ABB RAPID module: 000ACBDB

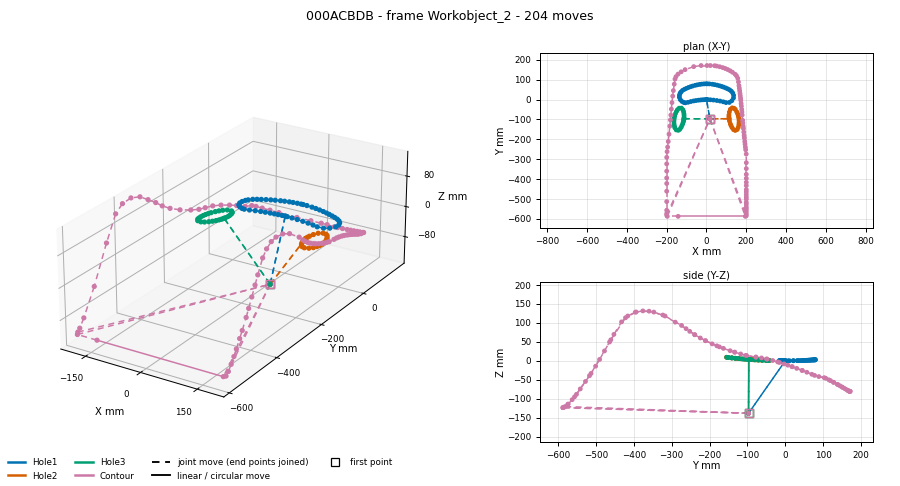
[picture p0: tool path of 000ACBDB in frame Workobject_2, 204 of 204 moves have a stored position in this frame; points joined in program order, loops and branches not executed]
MODULE Module1
        CONST robtarget Target_10:=[[26.851148837,-92.746056848,-137.743887933],[0.741188403,0.065864979,-0.059133334,0.6654358],[0,-1,-4,0],[9E+09,9E+09,9E+09,9E+09,9E+09,9E+09]];
    CONST robtarget H1_10:=[[5.822359777,-0.3029029,0.000239991],[0.999601623,-0.000118584,-0.000002778,-0.02822376],[0,-1,-1,0],[9E+09,9E+09,9E+09,9E+09,9E+09,9E+09]];
    CONST robtarget H1_20:=[[19.5237916,-1.229906178,0.000797071],[0.999216395,-0.000469719,-0.000020106,-0.039577455],[0,-1,0,0],[9E+09,9E+09,9E+09,9E+09,9E+09,9E+09]];
    CONST robtarget H1_30:=[[35.072112263,-2.692139723,0.003045649],[0.998507815,-0.001051706,-0.000057639,-0.054598844],[0,0,0,0],[9E+09,9E+09,9E+09,9E+09,9E+09,9E+09]];
    CONST robtarget H1_40:=[[51.872897494,-4.859700389,0.009441408],[0.997236669,-0.001878928,-0.000140271,-0.074266246],[0,0,0,0],[9E+09,9E+09,9E+09,9E+09,9E+09,9E+09]];
    CONST robtarget H1_50:=[[68.085842086,-7.671579778,0.023196339],[0.995164323,-0.002935794,-0.00030113,-0.098179733],[0,0,0,0],[9E+09,9E+09,9E+09,9E+09,9E+09,9E+09]];
    CONST robtarget H1_60:=[[84.016477696,-11.327527953,0.050315148],[0.991731899,-0.004378584,-0.000566998,-0.128251111],[0,0,0,0],[9E+09,9E+09,9E+09,9E+09,9E+09,9E+09]];
    CONST robtarget H1_70:=[[97.822312549,-15.342823644,0.092032674],[0.99493212,-0.005901634,-0.000604486,-0.100373712],[0,0,0,0],[9E+09,9E+09,9E+09,9E+09,9E+09,9E+09]];
    CONST robtarget H1_80:=[[114.627720719,-14.523229835,0.082502162],[0.982974748,-0.00555832,0.001038246,0.183653673],[0,0,0,0],[9E+09,9E+09,9E+09,9E+09,9E+09,9E+09]];
    CONST robtarget H1_90:=[[127.080680914,-6.164946714,0.015071505],[0.921910532,-0.002219077,0.0009341,0.387395372],[0,0,0,0],[9E+09,9E+09,9E+09,9E+09,9E+09,9E+09]];
    CONST robtarget H1_100:=[[135.46672126,7.649000487,0.023178554],[0.80179062,0.002410603,-0.00179684,0.597597492],[0,0,0,0],[9E+09,9E+09,9E+09,9E+09,9E+09,9E+09]];
    CONST robtarget H1_110:=[[136.157764084,21.042101165,0.174701099],[0.644801471,0.005362679,-0.006356556,0.764304847],[0,0,0,0],[9E+09,9E+09,9E+09,9E+09,9E+09,9E+09]];
    CONST robtarget H1_120:=[[131.874650789,32.837383759,0.404255936],[0.501756468,0.004666505,-0.008044466,0.864958934],[0,0,0,0],[9E+09,9E+09,9E+09,9E+09,9E+09,9E+09]];
    CONST robtarget H1_130:=[[124.935320592,41.709089606,0.620811537],[0.38373825,0.005805796,-0.013969102,0.923317991],[0,0,0,0],[9E+09,9E+09,9E+09,9E+09,9E+09,9E+09]];
    CONST robtarget H1_140:=[[116.229745208,48.490778985,0.856866002],[0.260536152,0.005127658,-0.018998209,0.965263533],[0,0,0,0],[9E+09,9E+09,9E+09,9E+09,9E+09,9E+09]];
    CONST robtarget H1_150:=[[106.531812126,53.651183132,1.078234714],[0.225840714,0.005240396,-0.022598239,0.973887997],[0,0,0,0],[9E+09,9E+09,9E+09,9E+09,9E+09,9E+09]];
    CONST robtarget H1_160:=[[96.895202054,58.051394326,1.295938149],[0.200438859,0.005260811,-0.025705853,0.979354786],[0,0,0,0],[9E+09,9E+09,9E+09,9E+09,9E+09,9E+09]];
    CONST robtarget H1_170:=[[86.200217498,62.31165247,1.532433666],[0.177271875,0.005181025,-0.02875481,0.983728113],[0,0,0,0],[9E+09,9E+09,9E+09,9E+09,9E+09,9E+09]];
    CONST robtarget H1_180:=[[76.71572938,65.636541326,1.734823668],[0.158973824,0.005020732,-0.031165772,0.986777994],[0,0,0,0],[9E+09,9E+09,9E+09,9E+09,9E+09,9E+09]];
    CONST robtarget H1_190:=[[65.746053731,69.013152347,1.956481108],[0.13904105,0.004727267,-0.033645532,0.989703601],[0,0,0,0],[9E+09,9E+09,9E+09,9E+09,9E+09,9E+09]];
    CONST robtarget H1_200:=[[53.528960273,72.219165213,2.182137232],[0.117236878,0.004256713,-0.036032694,0.99244095],[0,0,0,0],[9E+09,9E+09,9E+09,9E+09,9E+09,9E+09]];
    CONST robtarget H1_210:=[[41.391728548,74.836405126,2.377436106],[0.09495427,0.003628233,-0.038009225,0.994749125],[0,0,0,0],[9E+09,9E+09,9E+09,9E+09,9E+09,9E+09]];
    CONST robtarget H1_220:=[[29.543599616,76.831762317,2.533066199],[0.071726163,0.002844733,-0.039536532,0.996636407],[0,0,0,0],[9E+09,9E+09,9E+09,9E+09,9E+09,9E+09]];
    CONST robtarget H1_230:=[[14.423984972,78.513378499,2.668784241],[0.038405498,0.001570062,-0.040842603,0.998425978],[0,0,0,0],[9E+09,9E+09,9E+09,9E+09,9E+09,9E+09]];
    CONST robtarget H1_240:=[[3.529088415,79.053026073,2.713218089],[0.010521449,0.000436179,-0.041267795,0.999092627],[0,0,0,0],[9E+09,9E+09,9E+09,9E+09,9E+09,9E+09]];
    CONST robtarget H1_250:=[[-2.41393131,79.072935695,2.714873077],[0.007473374,0.000309011,0.041283579,-0.999119472],[-1,0,-2,0],[9E+09,9E+09,9E+09,9E+09,9E+09,9E+09]];
    CONST robtarget H1_260:=[[-12.79429846,78.631983773,2.678514834],[0.034459184,0.001412549,0.040935724,-0.99856639],[-1,0,-2,0],[9E+09,9E+09,9E+09,9E+09,9E+09,9E+09]];
    CONST robtarget H1_270:=[[-24.249294402,77.535857479,2.589375882],[0.060604597,0.002435338,0.04008087,-0.997353837],[-1,0,-2,0],[9E+09,9E+09,9E+09,9E+09,9E+09,9E+09]];
    CONST robtarget H1_280:=[[-34.022487008,76.144299483,2.478783806],[0.080709455,0.003161608,0.039008163,-0.995969051],[-1,0,-2,0],[9E+09,9E+09,9E+09,9E+09,9E+09,9E+09]];
    CONST robtarget H1_290:=[[-46.078360434,73.893089687,2.305893098],[0.103704766,0.003891012,0.037293549,-0.993901088],[-1,0,-2,0],[9E+09,9E+09,9E+09,9E+09,9E+09,9E+09]];
    CONST robtarget H1_300:=[[-56.338244037,71.532430973,2.132551125],[0.12227693,0.004378833,0.035518358,-0.991850606],[-1,0,-2,0],[9E+09,9E+09,9E+09,9E+09,9E+09,9E+09]];
    CONST robtarget H1_310:=[[-69.339991697,67.960014478,1.885584593],[0.145492672,0.004836435,0.032868463,-0.988801373],[-1,0,-2,0],[9E+09,9E+09,9E+09,9E+09,9E+09,9E+09]];
    CONST robtarget H1_320:=[[-80.066156183,64.506655976,1.664288351],[0.165267796,0.005087248,0.030343309,-0.985768715],[-1,0,-2,0],[9E+09,9E+09,9E+09,9E+09,9E+09,9E+09]];
    CONST robtarget H1_330:=[[-91.064867974,60.445719882,1.42572312],[0.187354774,0.005230691,0.027414242,-0.981895762],[-1,0,-2,0],[9E+09,9E+09,9E+09,9E+09,9E+09,9E+09]];
    CONST robtarget H1_340:=[[-101.905940758,55.839614159,1.18312319],[0.212963875,0.005260152,0.02413793,-0.976747705],[-1,0,-2,0],[9E+09,9E+09,9E+09,9E+09,9E+09,9E+09]];
    CONST robtarget H1_350:=[[-111.354611608,51.195431258,0.968343063],[0.241468672,0.005196012,0.020879464,-0.970170052],[-1,0,-2,0],[9E+09,9E+09,9E+09,9E+09,9E+09,9E+09]];
    CONST robtarget H1_360:=[[-120.397291393,45.950711286,0.761205788],[0.279512614,0.005021911,0.017247524,-0.959973959],[-1,0,-2,0],[9E+09,9E+09,9E+09,9E+09,9E+09,9E+09]];
    CONST robtarget H1_370:=[[-128.598391018,37.638733053,0.508601596],[0.433495604,0.005392781,0.011207446,-0.901069849],[-1,0,-2,0],[9E+09,9E+09,9E+09,9E+09,9E+09,9E+09]];
    CONST robtarget H1_380:=[[-132.59535291,31.513908724,0.380771009],[0.519470782,0.004385873,0.007214063,-0.854446504],[-1,0,-2,0],[9E+09,9E+09,9E+09,9E+09,9E+09,9E+09]];
    CONST robtarget H1_390:=[[-136.029541122,21.745014519,0.186590065],[0.636693593,0.005473624,0.006628875,-0.771068977],[-1,0,-2,0],[9E+09,9E+09,9E+09,9E+09,9E+09,9E+09]];
    CONST robtarget H1_400:=[[-136.249962901,11.059124977,0.04827139],[0.761868919,0.003316184,0.002819313,-0.647716609],[-1,0,-2,0],[9E+09,9E+09,9E+09,9E+09,9E+09,9E+09]];
    CONST robtarget H1_410:=[[-131.64005613,-0.499314804,0.000306325],[0.879140299,-0.000171436,-0.000093084,-0.476563004],[-1,0,-2,0],[9E+09,9E+09,9E+09,9E+09,9E+09,9E+09]];
    CONST robtarget H1_420:=[[-123.455867891,-9.420071732,0.0348798],[0.944806429,-0.003471167,-0.00120507,-0.327608472],[0,0,0,0],[9E+09,9E+09,9E+09,9E+09,9E+09,9E+09]];
    CONST robtarget H1_430:=[[-113.576963132,-14.907418805,0.086903996],[0.986261821,-0.005723499,-0.000957591,-0.165087688],[0,0,0,0],[9E+09,9E+09,9E+09,9E+09,9E+09,9E+09]];
    CONST robtarget H1_440:=[[-106.317369492,-16.310941036,0.103957245],[0.999811227,-0.006344693,-0.000116729,-0.018364159],[0,0,0,0],[9E+09,9E+09,9E+09,9E+09,9E+09,9E+09]];
    CONST robtarget H1_450:=[[-92.832473373,-13.839947638,0.074955681],[0.988817126,-0.005329902,0.000803336,0.149035693],[0,0,0,0],[9E+09,9E+09,9E+09,9E+09,9E+09,9E+09]];
    CONST robtarget H1_460:=[[-78.807083419,-10.018549669,0.039414696],[0.993068241,-0.003881094,0.000459005,0.117474235],[0,0,0,0],[9E+09,9E+09,9E+09,9E+09,9E+09,9E+09]];
    CONST robtarget H1_470:=[[-65.187150671,-7.109105356,0.019965876],[0.995622128,-0.00276447,0.000259127,0.093428411],[0,0,0,0],[9E+09,9E+09,9E+09,9E+09,9E+09,9E+09]];
    CONST robtarget H1_480:=[[-53.308517932,-5.077796928,0.010293707],[0.99709043,-0.001979187,0.000151084,0.076201937],[0,0,0,0],[9E+09,9E+09,9E+09,9E+09,9E+09,9E+09]];
    CONST robtarget H2_10:=[[113.353839197,-96.530340155,3.554586283],[0.748476702,-0.027164205,-0.024031886,-0.66216856],[0,-2,0,0],[9E+09,9E+09,9E+09,9E+09,9E+09,9E+09]];
    CONST robtarget H2_20:=[[115.464244857,-108.261236654,4.456832066],[0.783370795,-0.031725245,-0.025118376,-0.620236063],[0,-2,0,0],[9E+09,9E+09,9E+09,9E+09,9E+09,9E+09]];
    CONST robtarget H2_30:=[[119.841770859,-122.609627571,5.694437701],[0.820338947,-0.037394525,-0.025986049,-0.570061739],[0,-2,0,0],[9E+09,9E+09,9E+09,9E+09,9E+09,9E+09]];
    CONST robtarget H2_40:=[[123.527187524,-131.471644624,6.531828825],[0.840093436,-0.040906802,-0.026306691,-0.540256985],[0,-2,0,0],[9E+09,9E+09,9E+09,9E+09,9E+09,9E+09]];
    CONST robtarget H2_50:=[[128.497488384,-141.378498828,7.628466543],[0.858996843,-0.051948016,-0.030746201,-0.508409774],[0,-2,0,0],[9E+09,9E+09,9E+09,9E+09,9E+09,9E+09]];
    CONST robtarget H2_60:=[[136.105023801,-151.417458815,8.807259628],[0.9370628,-0.052968209,-0.019477183,-0.344569757],[0,-2,1,0],[9E+09,9E+09,9E+09,9E+09,9E+09,9E+09]];
    CONST robtarget H2_70:=[[144.44174435,-155.241358627,9.235032257],[0.998005294,-0.054882138,-0.001713201,-0.031152033],[0,-2,1,0],[9E+09,9E+09,9E+09,9E+09,9E+09,9E+09]];
    CONST robtarget H2_80:=[[154.006118475,-150.661083946,8.721245568],[0.908752155,-0.051640643,0.023496208,0.41346184],[0,-2,-2,0],[9E+09,9E+09,9E+09,9E+09,9E+09,9E+09]];
    CONST robtarget H2_90:=[[159.658512318,-139.997126678,7.46002746],[0.79556302,-0.048534782,0.036779081,0.60280275],[0,-2,-2,0],[9E+09,9E+09,9E+09,9E+09,9E+09,9E+09]];
    CONST robtarget H2_100:=[[162.376179916,-127.516765295,6.151270714],[0.758777117,-0.035896886,0.030733454,0.649633862],[0,-2,-2,0],[9E+09,9E+09,9E+09,9E+09,9E+09,9E+09]];
    CONST robtarget H2_110:=[[163.475309343,-117.188024925,5.209561495],[0.726089453,-0.031708487,0.029967159,0.686214724],[0,-2,-2,0],[9E+09,9E+09,9E+09,9E+09,9E+09,9E+09]];
    CONST robtarget H2_120:=[[163.492051849,-105.498676679,4.235442415],[0.68742213,-0.02716136,0.028653424,0.725184154],[0,-2,-2,0],[9E+09,9E+09,9E+09,9E+09,9E+09,9E+09]];
    CONST robtarget H2_130:=[[162.227653576,-93.852494517,3.362554996],[0.647198475,-0.022863035,0.026901004,0.761503612],[0,-2,-2,0],[9E+09,9E+09,9E+09,9E+09,9E+09,9E+09]];
    CONST robtarget H2_140:=[[160.115266627,-83.883832167,2.693495802],[0.611329591,-0.019384569,0.025073576,0.790741226],[0,-2,-2,0],[9E+09,9E+09,9E+09,9E+09,9E+09,9E+09]];
    CONST robtarget H2_150:=[[156.297628088,-71.997621841,1.990746535],[0.566564132,-0.015498139,0.022528309,0.823563821],[0,-2,-2,0],[9E+09,9E+09,9E+09,9E+09,9E+09,9E+09]];
    CONST robtarget H2_160:=[[151.695554905,-61.57696201,1.460402668],[0.525052814,-0.012338693,0.019992429,0.850745321],[0,-2,-2,0],[9E+09,9E+09,9E+09,9E+09,9E+09,9E+09]];
    CONST robtarget H2_170:=[[144.697582417,-49.505236902,0.947141756],[0.473504531,-0.008991922,0.016722668,0.880586711],[0,-2,-2,0],[9E+09,9E+09,9E+09,9E+09,9E+09,9E+09]];
    CONST robtarget H2_180:=[[138.479508342,-43.903121696,0.746107759],[0.27767732,-0.00468769,0.016215326,0.960526103],[0,-2,-2,0],[9E+09,9E+09,9E+09,9E+09,9E+09,9E+09]];
    CONST robtarget H2_190:=[[129.228972872,-41.777368956,0.676021991],[0.096272542,-0.00154838,-0.016002122,-0.995225167],[0,-2,-1,0],[9E+09,9E+09,9E+09,9E+09,9E+09,9E+09]];
    CONST robtarget H2_200:=[[119.969352837,-48.884343518,0.92369665],[0.471525813,-0.008844606,-0.016537415,-0.88165282],[0,-2,-1,0],[9E+09,9E+09,9E+09,9E+09,9E+09,9E+09]];
    CONST robtarget H2_210:=[[114.862919521,-62.738334039,1.515519436],[0.627584743,-0.01501889,-0.018622826,-0.778180579],[0,-2,0,0],[9E+09,9E+09,9E+09,9E+09,9E+09,9E+09]];
    CONST robtarget H2_220:=[[112.782345249,-77.613018099,2.309812122],[0.68393145,-0.020117567,-0.021445948,-0.728953446],[0,-2,0,0],[9E+09,9E+09,9E+09,9E+09,9E+09,9E+09]];
    CONST robtarget H2_230:=[[112.619785188,-86.868177001,2.886201345],[0.71669986,-0.023502264,-0.022847584,-0.69661104],[0,-2,0,0],[9E+09,9E+09,9E+09,9E+09,9E+09,9E+09]];
    CONST robtarget H2_240:=[[-146.211495519,-51.850497933,1.03831773],[0.483686197,-0.009610968,-0.017386784,-0.875015995],[0,0,0,0],[9E+09,9E+09,9E+09,9E+09,9E+09,9E+09]];
    CONST robtarget H2_250:=[[-149.107034596,-56.713931894,1.240531943],[0.504739909,-0.010947301,-0.018717571,-0.862999092],[0,0,0,0],[9E+09,9E+09,9E+09,9E+09,9E+09,9E+09]];
    CONST robtarget H2_260:=[[-151.196381116,-60.595266341,1.414599226],[0.521004601,-0.012053404,-0.019739665,-0.853240451],[0,0,0,0],[9E+09,9E+09,9E+09,9E+09,9E+09,9E+09]];
    CONST robtarget H2_270:=[[-153.664684888,-65.700778492,1.660655818],[0.541786795,-0.013561095,-0.021028685,-0.840143416],[0,0,0,0],[9E+09,9E+09,9E+09,9E+09,9E+09,9E+09]];
    CONST robtarget H2_280:=[[-155.154121582,-69.132687567,1.836925418],[0.555398018,-0.014605886,-0.021858445,-0.831169007],[0,0,0,0],[9E+09,9E+09,9E+09,9E+09,9E+09,9E+09]];
    CONST robtarget H2_290:=[[-156.838393073,-73.438168646,2.070385804],[0.572126761,-0.015952496,-0.022858608,-0.819691388],[0,0,0,0],[9E+09,9E+09,9E+09,9E+09,9E+09,9E+09]];
    CONST robtarget H2_300:=[[-158.385938506,-77.933906529,2.328748906],[0.589243008,-0.01740327,-0.023847263,-0.807416318],[0,0,0,0],[9E+09,9E+09,9E+09,9E+09,9E+09,9E+09]];
    CONST robtarget H2_310:=[[-159.957660119,-83.287580126,2.655778618],[0.609137583,-0.019181563,-0.024956614,-0.792439676],[0,0,0,0],[9E+09,9E+09,9E+09,9E+09,9E+09,9E+09]];
    CONST robtarget H2_320:=[[-160.980080082,-87.442702976,2.924049197],[0.624309267,-0.020604348,-0.025759704,-0.780480517],[0,0,0,0],[9E+09,9E+09,9E+09,9E+09,9E+09,9E+09]];
    CONST robtarget H2_330:=[[-161.982296625,-92.416885735,3.261751009],[0.642117861,-0.022350365,-0.026655965,-0.765816279],[0,0,0,0],[9E+09,9E+09,9E+09,9E+09,9E+09,9E+09]];
    CONST robtarget H2_340:=[[-162.658869303,-96.728725981,3.569023092],[0.657295549,-0.023901838,-0.027373156,-0.752756252],[0,0,0,0],[9E+09,9E+09,9E+09,9E+09,9E+09,9E+09]];
    CONST robtarget H2_350:=[[-163.3089721,-102.754467741,4.020957585],[0.678104452,-0.026127054,-0.028278994,-0.73395642],[0,0,0,0],[9E+09,9E+09,9E+09,9E+09,9E+09,9E+09]];
    CONST robtarget H2_360:=[[-163.588731895,-107.752945715,4.415691555],[0.695018407,-0.028020761,-0.028942698,-0.717862501],[0,0,0,0],[9E+09,9E+09,9E+09,9E+09,9E+09,9E+09]];
    CONST robtarget H2_370:=[[-163.618228194,-113.559417795,4.896727938],[0.714282559,-0.030273854,-0.029608796,-0.698575149],[0,0,0,0],[9E+09,9E+09,9E+09,9E+09,9E+09,9E+09]];
    CONST robtarget H2_380:=[[-163.400274185,-118.383550137,5.314692806],[0.729948009,-0.032185694,-0.030075106,-0.68208172],[0,0,0,0],[9E+09,9E+09,9E+09,9E+09,9E+09,9E+09]];
    CONST robtarget H2_390:=[[-162.725296292,-125.102597289,5.924399836],[0.751271747,-0.034905156,-0.030588292,-0.658359133],[0,0,0,0],[9E+09,9E+09,9E+09,9E+09,9E+09,9E+09]];
    CONST robtarget H2_400:=[[-161.284238305,-133.391691812,6.720562185],[0.776702072,-0.038351334,-0.030988752,-0.627935318],[0,0,0,0],[9E+09,9E+09,9E+09,9E+09,9E+09,9E+09]];
    CONST robtarget H2_410:=[[-159.646201857,-140.03915335,7.465181503],[0.795699451,-0.048528933,-0.036759329,-0.602624326],[0,0,0,0],[9E+09,9E+09,9E+09,9E+09,9E+09,9E+09]];
    CONST robtarget H2_420:=[[-157.038646765,-146.326115351,8.219442761],[0.863010837,-0.050522948,-0.029376394,-0.501793537],[0,0,0,0],[9E+09,9E+09,9E+09,9E+09,9E+09,9E+09]];
    CONST robtarget H2_430:=[[-154.143947087,-150.501789747,8.703078987],[0.906591242,-0.051576054,-0.023790201,-0.418170129],[0,0,0,0],[9E+09,9E+09,9E+09,9E+09,9E+09,9E+09]];
    CONST robtarget H2_440:=[[-151.052306188,-153.326067118,9.022258344],[0.953526504,-0.053170779,-0.016512614,-0.296120598],[0,0,0,0],[9E+09,9E+09,9E+09,9E+09,9E+09,9E+09]];
    CONST robtarget H2_450:=[[-147.24920751,-155.018200209,9.210400641],[0.992262537,-0.054655516,-0.006130652,-0.111311491],[-1,1,-2,0],[9E+09,9E+09,9E+09,9E+09,9E+09,9E+09]];
    CONST robtarget H2_460:=[[-141.774746784,-154.730898904,9.178619755],[0.986433645,-0.054448707,0.008535421,0.154632303],[-1,1,-2,0],[9E+09,9E+09,9E+09,9E+09,9E+09,9E+09]];
    CONST robtarget H2_470:=[[-137.124498645,-152.232288983,8.899410279],[0.946429998,-0.053189584,0.017871487,0.317996442],[-1,1,-2,0],[9E+09,9E+09,9E+09,9E+09,9E+09,9E+09]];
    CONST robtarget H2_480:=[[-133.464165375,-148.877446335,8.516599917],[0.914460182,-0.052613853,0.02304735,0.400578554],[-1,1,-2,0],[9E+09,9E+09,9E+09,9E+09,9E+09,9E+09]];
    CONST robtarget H2_490:=[[-130.178716496,-144.342311293,7.984808374],[0.86461459,-0.051289546,0.029597151,0.498933866],[0,0,0,0],[9E+09,9E+09,9E+09,9E+09,9E+09,9E+09]];
    CONST robtarget H2_500:=[[-127.259861509,-139.094676901,7.34918768],[0.854541306,-0.052433266,0.031646215,0.515760047],[0,0,0,0],[9E+09,9E+09,9E+09,9E+09,9E+09,9E+09]];
    CONST robtarget H2_510:=[[-126.560241996,-137.75989446,7.184074667],[0.851876838,-0.052707296,0.032178927,0.520088753],[0,0,0,0],[9E+09,9E+09,9E+09,9E+09,9E+09,9E+09]];
    CONST robtarget H2_520:=[[-124.896955353,-134.374624635,6.818180126],[0.846081591,-0.042055694,0.026381033,0.530736565],[0,0,0,0],[9E+09,9E+09,9E+09,9E+09,9E+09,9E+09]];
    CONST robtarget H2_530:=[[-122.756510357,-129.759645709,6.365744431],[0.836453631,-0.040228874,0.026256095,0.545928181],[0,0,0,0],[9E+09,9E+09,9E+09,9E+09,9E+09,9E+09]];
    CONST robtarget H3_90:=[[-151.032520543,-60.277726678,1.399936408],[0.519689718,-0.011961435,-0.019657661,-0.854045138],[-1,1,1,0],[9E+09,9E+09,9E+09,9E+09,9E+09,9E+09]];
    CONST robtarget H3_100:=[[-155.411707479,-69.759012426,1.870035967],[0.557852374,-0.014799042,-0.022007461,-0.829516358],[-1,1,1,0],[9E+09,9E+09,9E+09,9E+09,9E+09,9E+09]];
    CONST robtarget H3_110:=[[-159.625213408,-82.068644739,2.579473667],[0.604642285,-0.018772206,-0.024709982,-0.79589241],[-1,1,1,0],[9E+09,9E+09,9E+09,9E+09,9E+09,9E+09]];
    CONST robtarget H3_120:=[[-161.878029858,-91.838551641,3.22156317],[0.640063811,-0.022144937,-0.026555455,-0.767543306],[-1,1,1,0],[9E+09,9E+09,9E+09,9E+09,9E+09,9E+09]];
    CONST robtarget H3_130:=[[-163.203180759,-101.514565736,3.925825431],[0.673850412,-0.025662667,-0.028101558,-0.737887087],[-1,1,1,0],[9E+09,9E+09,9E+09,9E+09,9E+09,9E+09]];
    CONST robtarget H3_140:=[[-163.644574839,-111.272609544,4.704398344],[0.706753039,-0.029380699,-0.02935936,-0.706240005],[-1,1,1,0],[9E+09,9E+09,9E+09,9E+09,9E+09,9E+09]];
    CONST robtarget H3_150:=[[-163.073115646,-122.1735858,5.654675757],[0.742058033,-0.033712272,-0.030383983,-0.668797556],[-1,1,1,0],[9E+09,9E+09,9E+09,9E+09,9E+09,9E+09]];
    CONST robtarget H3_160:=[[-161.45041585,-132.605221729,6.642943788],[0.774331563,-0.038018965,-0.030963091,-0.630877544],[0,0,0,0],[9E+09,9E+09,9E+09,9E+09,9E+09,9E+09]];
    CONST robtarget H3_170:=[[-159.100531555,-141.897037426,7.691315566],[0.801095296,-0.048179165,-0.035972301,-0.5955091],[0,0,0,0],[9E+09,9E+09,9E+09,9E+09,9E+09,9E+09]];
    CONST robtarget H3_180:=[[-152.159173857,-152.48346178,8.927706865],[0.937417285,-0.05258876,-0.01927966,-0.34367361],[0,0,0,0],[9E+09,9E+09,9E+09,9E+09,9E+09,9E+09]];
    CONST robtarget H3_190:=[[-141.819169103,-154.744996081,9.180180698],[0.986731419,-0.054459539,0.008429136,0.152722671],[-1,1,-2,0],[9E+09,9E+09,9E+09,9E+09,9E+09,9E+09]];
    CONST robtarget H3_200:=[[-134.593857995,-150.038962909,8.65016057],[0.923763552,-0.052723447,0.021614172,0.378700364],[-1,1,-2,0],[9E+09,9E+09,9E+09,9E+09,9E+09,9E+09]];
    CONST robtarget H3_210:=[[-128.24945161,-140.928737155,7.573794657],[0.858129871,-0.052045202,0.030922266,0.509851189],[0,0,0,0],[9E+09,9E+09,9E+09,9E+09,9E+09,9E+09]];
    CONST robtarget H3_220:=[[-123.697125678,-131.841961932,6.568031258],[0.840871704,-0.041053612,0.026317047,0.539033201],[0,0,0,0],[9E+09,9E+09,9E+09,9E+09,9E+09,9E+09]];
    CONST robtarget H3_230:=[[-119.718209049,-122.278505657,5.664229892],[0.819556015,-0.037263357,0.025971018,0.571196014],[0,0,0,0],[9E+09,9E+09,9E+09,9E+09,9E+09,9E+09]];
    CONST robtarget H3_240:=[[-116.914843491,-113.780868438,4.915548572],[0.79834197,-0.033899897,0.025507908,0.600708118],[0,0,0,0],[9E+09,9E+09,9E+09,9E+09,9E+09,9E+09]];
    CONST robtarget H3_250:=[[-115.129078785,-106.801898067,4.339203478],[0.779261299,-0.031153062,0.025003039,0.625424786],[0,0,0,0],[9E+09,9E+09,9E+09,9E+09,9E+09,9E+09]];
    CONST robtarget H3_260:=[[-113.89814797,-100.37190359,3.839131682],[0.760357658,-0.02864585,0.024428314,0.648412603],[0,0,0,0],[9E+09,9E+09,9E+09,9E+09,9E+09,9E+09]];
    CONST robtarget H3_270:=[[-2.8649147,79.065647891,2.714269653],[0.008725056,0.000360634,0.041277791,-0.999109547],[0,0,0,0],[9E+09,9E+09,9E+09,9E+09,9E+09,9E+09]];
    CONST robtarget H3_280:=[[-6.334685984,78.972502416,2.706566926],[0.018106651,0.000746596,0.041203984,-0.998986398],[-1,0,-2,0],[9E+09,9E+09,9E+09,9E+09,9E+09,9E+09]];
    CONST robtarget H3_290:=[[-10.115541125,78.798786754,2.692234704],[0.027838843,0.001144817,0.041066905,-0.99876784],[-1,0,-2,0],[9E+09,9E+09,9E+09,9E+09,9E+09,9E+09]];
    CONST robtarget H3_300:=[[-12.967121471,78.620009059,2.677531525],[0.034878932,0.001429434,0.040926321,-0.998552178],[-1,0,-2,0],[9E+09,9E+09,9E+09,9E+09,9E+09,9E+09]];
    CONST robtarget H3_310:=[[-17.148960654,78.286603961,2.650238016],[0.044763067,0.001824202,0.040665248,-0.998167961],[-1,0,-2,0],[9E+09,9E+09,9E+09,9E+09,9E+09,9E+09]];
    CONST robtarget H3_320:=[[-21.565389337,77.846298964,2.614439805],[0.054738413,0.002212749,0.040322016,-0.99768379],[-1,0,-2,0],[9E+09,9E+09,9E+09,9E+09,9E+09,9E+09]];
    CONST robtarget H3_330:=[[-27.10271187,77.171238947,2.56012345],[0.066674643,0.002660905,0.039798533,-0.996977175],[-1,0,-2,0],[9E+09,9E+09,9E+09,9E+09,9E+09,9E+09]];
    CONST robtarget H3_340:=[[-30.430871342,76.702094493,2.522774606],[0.073533349,0.002909696,0.039436657,-0.99650847],[-1,0,-2,0],[9E+09,9E+09,9E+09,9E+09,9E+09,9E+09]];
    CONST robtarget H3_350:=[[-36.071948771,75.802452022,2.452048787],[0.084738305,0.003298132,0.038746269,-0.995644148],[-1,0,-2,0],[9E+09,9E+09,9E+09,9E+09,9E+09,9E+09]];
    CONST robtarget H3_360:=[[-40.871398594,74.935924168,2.385053721],[0.093983304,0.003597617,0.038084851,-0.99483855],[-1,0,-2,0],[9E+09,9E+09,9E+09,9E+09,9E+09,9E+09]];
    CONST robtarget H3_370:=[[-45.168917683,74.082828858,2.320177807],[0.102030362,0.003842105,0.03743714,-0.994069165],[-1,0,-2,0],[9E+09,9E+09,9E+09,9E+09,9E+09,9E+09]];
    CONST robtarget H3_380:=[[-50.551705589,72.913466151,2.232974457],[0.111870475,0.004118016,0.036554348,-0.9930417],[-1,0,-2,0],[9E+09,9E+09,9E+09,9E+09,9E+09,9E+09]];
    CONST robtarget H3_390:=[[-55.549209342,71.72828369,2.146624137],[0.12086579,0.004345406,0.035664857,-0.992018445],[-1,0,-2,0],[9E+09,9E+09,9E+09,9E+09,9E+09,9E+09]];
    CONST robtarget H3_400:=[[-61.927505303,70.076739745,2.029695738],[0.132245008,0.004596819,0.034433562,-0.990608125],[-1,0,-2,0],[9E+09,9E+09,9E+09,9E+09,9E+09,9E+09]];
    CONST robtarget H3_410:=[[-68.62429444,68.173796841,1.899846076],[0.144200224,0.004815742,0.033025964,-0.988985536],[-1,0,-2,0],[9E+09,9E+09,9E+09,9E+09,9E+09,9E+09]];
    CONST robtarget H3_420:=[[-73.053957234,66.817667973,1.810494492],[0.152245741,0.004935728,0.032029173,-0.987811219],[-1,0,-2,0],[9E+09,9E+09,9E+09,9E+09,9E+09,9E+09]];
    CONST robtarget H3_430:=[[-79.167968195,64.814210939,1.683307668],[0.163563945,0.005070503,0.030566866,-0.98604604],[-1,0,-2,0],[9E+09,9E+09,9E+09,9E+09,9E+09,9E+09]];
    CONST robtarget H3_440:=[[-84.238390617,63.031729667,1.574946041],[0.173348853,0.005155043,0.029274559,-0.984411804],[-1,0,-2,0],[9E+09,9E+09,9E+09,9E+09,9E+09,9E+09]];
    CONST robtarget H3_450:=[[-88.890544547,61.293706375,1.47361581],[0.182762993,0.005211361,0.028022536,-0.982743745],[-1,0,-2,0],[9E+09,9E+09,9E+09,9E+09,9E+09,9E+09]];
    CONST robtarget H3_460:=[[-95.479750625,58.649863335,1.327607794],[0.197052537,0.005258002,0.026132891,-0.980030471],[-1,0,-2,0],[9E+09,9E+09,9E+09,9E+09,9E+09,9E+09]];
    CONST robtarget H3_470:=[[-102.280879458,55.667700917,1.174643979],[0.213962984,0.0052591,0.024016447,-0.976532331],[-1,0,-2,0],[9E+09,9E+09,9E+09,9E+09,9E+09,9E+09]];
    CONST robtarget H3_480:=[[-108.13915594,52.85405221,1.041654244],[0.230734556,0.005228689,0.022039645,-0.972753042],[-1,0,-2,0],[9E+09,9E+09,9E+09,9E+09,9E+09,9E+09]];
    CONST robtarget H3_490:=[[-112.844891048,50.394720403,0.934303108],[0.246880393,0.005177668,0.020321316,-0.968819027],[-1,0,-2,0],[9E+09,9E+09,9E+09,9E+09,9E+09,9E+09]];
    CONST robtarget H3_500:=[[-118.347328888,47.230096261,0.808297005],[0.270328919,0.005090046,0.018124474,-0.962583955],[-1,0,-2,0],[9E+09,9E+09,9E+09,9E+09,9E+09,9E+09]];
    CONST robtarget H3_510:=[[-123.252061757,43.344922201,0.672097613],[0.369331386,0.005987744,0.015069422,-0.929156277],[-1,0,-2,0],[9E+09,9E+09,9E+09,9E+09,9E+09,9E+09]];
    CONST robtarget H3_520:=[[-127.934077654,38.449353154,0.529203927],[0.422392751,0.005479549,0.011756156,-0.906320104],[-1,0,-2,0],[9E+09,9E+09,9E+09,9E+09,9E+09,9E+09]];
    CONST robtarget H3_530:=[[-130.333027831,35.297380543,0.453953091],[0.466730019,0.005087182,0.009640709,-0.884332667],[-1,0,-2,0],[9E+09,9E+09,9E+09,9E+09,9E+09,9E+09]];
    CONST robtarget H3_540:=[[-132.17837315,32.294925109,0.39435499],[0.509131796,0.004556015,0.007701531,-0.860642053],[-1,0,-2,0],[9E+09,9E+09,9E+09,9E+09,9E+09,9E+09]];
    CONST robtarget H3_550:=[[-134.71177698,26.636386283,0.280260541],[0.579626455,0.006116566,0.008598406,-0.814813984],[-1,0,-2,0],[9E+09,9E+09,9E+09,9E+09,9E+09,9E+09]];
    CONST robtarget H3_560:=[[-135.896350855,22.401538281,0.198051061],[0.629116362,0.005573246,0.006885644,-0.777260657],[-1,0,-2,0],[9E+09,9E+09,9E+09,9E+09,9E+09,9E+09]];
    CONST robtarget H3_570:=[[-136.601751104,16.725219048,0.110313821],[0.694946599,0.004587102,0.004742989,-0.719031075],[-1,0,-2,0],[9E+09,9E+09,9E+09,9E+09,9E+09,9E+09]];
    CONST robtarget H3_580:=[[-136.364426363,11.829196267,0.055209838],[0.752707235,0.003505804,0.003065878,-0.658338916],[-1,0,-2,0],[9E+09,9E+09,9E+09,9E+09,9E+09,9E+09]];
    CONST robtarget H3_590:=[[-135.317213939,7.16505842,0.020360477],[0.807113502,0.002275064,0.001660903,-0.590389584],[-1,0,-2,0],[9E+09,9E+09,9E+09,9E+09,9E+09,9E+09]];
    CONST robtarget H3_600:=[[-133.896828693,3.546037028,0.005139696],[0.843810747,0.001174085,0.000746546,-0.536639067],[-1,0,-2,0],[9E+09,9E+09,9E+09,9E+09,9E+09,9E+09]];
    CONST robtarget H3_610:=[[-132.499178413,0.890292813,0.000520082],[0.867590512,0.000302632,0.000173423,-0.497279179],[-1,0,-2,0],[9E+09,9E+09,9E+09,9E+09,9E+09,9E+09]];
    CONST robtarget H3_620:=[[-129.838126372,-3.018698325,0.003774958],[0.898911267,-0.001061336,-0.000518189,-0.438129134],[-1,0,-2,0],[9E+09,9E+09,9E+09,9E+09,9E+09,9E+09]];
    CONST robtarget H3_630:=[[-127.070682613,-6.174541253,0.015118447],[0.921963416,-0.002224304,-0.000934287,-0.387269466],[-1,0,-2,0],[9E+09,9E+09,9E+09,9E+09,9E+09,9E+09]];
    CONST robtarget H3_640:=[[-123.852197312,-9.103311942,0.032589879],[0.942578351,-0.00334709,-0.001187192,-0.333966224],[0,0,0,0],[9E+09,9E+09,9E+09,9E+09,9E+09,9E+09]];
    CONST robtarget H3_650:=[[-119.78104127,-11.972585089,0.056175177],[0.963078526,-0.004491085,-0.00125712,-0.269180243],[0,0,0,0],[9E+09,9E+09,9E+09,9E+09,9E+09,9E+09]];
    CONST robtarget H3_660:=[[-114.892244394,-14.41917797,0.08133014],[0.982105326,-0.005513536,-0.001057005,-0.188248805],[0,0,0,0],[9E+09,9E+09,9E+09,9E+09,9E+09,9E+09]];
    CONST robtarget H3_670:=[[-110.529824325,-15.766113082,0.097156934],[0.994171715,-0.006096159,-0.000660851,-0.10763364],[0,0,0,0],[9E+09,9E+09,9E+09,9E+09,9E+09,9E+09]];
    CONST robtarget H3_680:=[[-106.636993824,-16.296877303,0.103778698],[0.999652295,-0.006338058,-0.000162455,-0.025594776],[0,0,0,0],[9E+09,9E+09,9E+09,9E+09,9E+09,9E+09]];
    CONST robtarget H3_690:=[[-102.556213296,-16.14770427,0.101894628],[0.998368294,-0.006227435,0.000358422,0.056761259],[0,0,0,0],[9E+09,9E+09,9E+09,9E+09,9E+09,9E+09]];
    CONST robtarget H3_700:=[[-99.223184663,-15.620755469,0.095381381],[0.995527055,-0.006012115,0.000576944,0.094283639],[0,0,0,0],[9E+09,9E+09,9E+09,9E+09,9E+09,9E+09]];
    CONST robtarget H3_710:=[[-94.170932178,-14.257928738,0.079529473],[0.988278205,-0.005486906,0.000847049,0.152562661],[0,0,0,0],[9E+09,9E+09,9E+09,9E+09,9E+09,9E+09]];
    CONST robtarget H3_720:=[[-90.175727328,-13.04018978,0.066581385],[0.989797444,-0.005028604,0.000723503,0.142391046],[0,0,0,0],[9E+09,9E+09,9E+09,9E+09,9E+09,9E+09]];
    CONST robtarget H3_730:=[[-86.658854429,-12.039206106,0.056798518],[0.990955715,-0.004649767,0.000629221,0.134107251],[0,0,0,0],[9E+09,9E+09,9E+09,9E+09,9E+09,9E+09]];
    CONST robtarget H3_740:=[[-80.714319729,-10.483924035,0.043136871],[0.99260646,-0.004058789,0.00049634,0.121308269],[0,0,0,0],[9E+09,9E+09,9E+09,9E+09,9E+09,9E+09]];
    CONST robtarget H3_750:=[[-77.410247014,-9.687464385,0.036870096],[0.993387613,-0.003753893,0.000433373,0.114746548],[0,0,0,0],[9E+09,9E+09,9E+09,9E+09,9E+09,9E+09]];
    CONST robtarget H3_760:=[[-72.383449699,-8.560552597,0.028848458],[0.994416059,-0.003322868,0.000352678,0.10547766],[0,0,0,0],[9E+09,9E+09,9E+09,9E+09,9E+09,9E+09]];
    CONST robtarget H3_770:=[[-67.562878304,-7.56835607,0.022597737],[0.995254538,-0.002941456,0.000287499,0.09726083],[0,0,0,0],[9E+09,9E+09,9E+09,9E+09,9E+09,9E+09]];
    CONST robtarget H3_780:=[[-63.463310256,-6.787553886,0.018221683],[0.995871354,-0.002640417,0.000240217,0.09073707],[0,0,0,0],[9E+09,9E+09,9E+09,9E+09,9E+09,9E+09]];
    CONST robtarget H3_790:=[[-59.51784174,-6.086891977,0.014698091],[0.996391091,-0.002369867,0.000202028,0.08484773],[0,0,0,0],[9E+09,9E+09,9E+09,9E+09,9E+09,9E+09]];
    CONST robtarget H3_800:=[[-54.202065001,-5.216273397,0.010850686],[0.996997972,-0.002032872,0.000157723,0.077400821],[0,0,0,0],[9E+09,9E+09,9E+09,9E+09,9E+09,9E+09]];
    CONST robtarget H3_810:=[[-50.771912193,-4.696500345,0.00883786],[0.997338978,-0.001831319,0.0001336,0.072880662],[0,0,0,0],[9E+09,9E+09,9E+09,9E+09,9E+09,9E+09]];
    CONST robtarget H3_820:=[[-46.411369666,-4.080294062,0.006722909],[0.997722172,-0.001592048,0.00010779,0.067438276],[0,0,0,0],[9E+09,9E+09,9E+09,9E+09,9E+09,9E+09]];
    CONST robtarget H3_830:=[[-42.861068035,-3.613542485,0.005317609],[0.997998771,-0.001410633,0.000089349,0.063217521],[0,0,0,0],[9E+09,9E+09,9E+09,9E+09,9E+09,9E+09]];
    CONST robtarget H3_840:=[[-38.453966225,-3.075514751,0.00391081],[0.998302162,-0.001201226,0.000069922,0.058235261],[0,0,0,0],[9E+09,9E+09,9E+09,9E+09,9E+09,9E+09]];
    CONST robtarget H3_850:=[[-34.755015713,-2.657501891,0.002973119],[0.998526064,-0.00103825,0.000056553,0.054264346],[0,0,0,0],[9E+09,9E+09,9E+09,9E+09,9E+09,9E+09]];
    CONST robtarget H3_860:=[[-30.571371065,-2.219783885,0.002136992],[0.998750411,-0.00086771,0.000043405,0.049968604],[0,0,0,0],[9E+09,9E+09,9E+09,9E+09,9E+09,9E+09]];
    CONST robtarget H3_870:=[[-26.619058995,-1.838903801,0.00153256],[0.998936754,-0.000719067,0.000033069,0.046096023],[0,0,0,0],[9E+09,9E+09,9E+09,9E+09,9E+09,9E+09]];
    CONST robtarget H3_880:=[[-22.570276908,-1.480013088,0.001065682],[0.99910403,-0.000576332,0.000025025,0.042317897],[0,0,0,0],[9E+09,9E+09,9E+09,9E+09,9E+09,9E+09]];
    CONST robtarget H3_890:=[[-18.120873762,-1.120361099,0.00069462],[0.999264525,-0.000420446,0.000018071,0.038343603],[0,0,0,0],[9E+09,9E+09,9E+09,9E+09,9E+09,9E+09]];
    CONST robtarget H3_900:=[[-13.977341342,-0.816811364,0.000461028],[0.999394539,-0.000288381,0.000012407,0.034791842],[0,0,0,0],[9E+09,9E+09,9E+09,9E+09,9E+09,9E+09]];
    CONST robtarget H3_910:=[[-9.744674824,-0.53665948,0.000313118],[0.999509625,-0.00018012,0.000007204,0.03131256],[0,0,0,0],[9E+09,9E+09,9E+09,9E+09,9E+09,9E+09]];
    CONST robtarget H3_920:=[[-5.685631557,-0.295203696,0.000238325],[0.999604622,-0.000099291,0.000003135,0.028117426],[0,0,0,0],[9E+09,9E+09,9E+09,9E+09,9E+09,9E+09]];
    CONST robtarget H3_930:=[[-2.455941119,-0.12133202,0.000213395],[0.999670366,-0.0000434,0.000000904,0.025674065],[0,0,0,0],[9E+09,9E+09,9E+09,9E+09,9E+09,9E+09]];
    CONST robtarget H3_940:=[[-0.399878518,-0.018777868,0.00020889],[0.999708001,0.000020089,0.000000752,0.024164258],[0,0,0,0],[9E+09,9E+09,9E+09,9E+09,9E+09,9E+09]];
    CONST robtarget H3_950:=[[1.088503446,-0.052412558,0.00020961],[0.999695741,0.000001267,-0.000000821,-0.024666274],[0,0,0,0],[9E+09,9E+09,9E+09,9E+09,9E+09,9E+09]];
    CONST robtarget H3_960:=[[3.551807296,-0.17853948,0.000219082],[0.999648966,-0.000062644,-0.000001528,-0.026494159],[0,0,0,0],[9E+09,9E+09,9E+09,9E+09,9E+09,9E+09]];
    CONST robtarget H3_970:=[[6.028972352,-0.31461269,0.000242588],[0.999597108,-0.000106704,-0.000003399,-0.028383282],[0,0,0,0],[9E+09,9E+09,9E+09,9E+09,9E+09,9E+09]];
    CONST robtarget H3_980:=[[8.054396824,-0.432934291,0.0002751],[0.999550909,-0.000146008,-0.000005318,-0.029965956],[0,0,0,0],[9E+09,9E+09,9E+09,9E+09,9E+09,9E+09]];
    CONST robtarget H3_990:=[[10.085122155,-0.558098182,0.000322142],[0.999500981,-0.000189832,-0.00000753,-0.031587218],[0,0,0,0],[9E+09,9E+09,9E+09,9E+09,9E+09,9E+09]];
    CONST robtarget H3_1000:=[[13.436624039,-0.77935711,0.00043748],[0.99941022,-0.00027503,-0.000011632,-0.034338564],[0,0,0,0],[9E+09,9E+09,9E+09,9E+09,9E+09,9E+09]];
    CONST robtarget H3_1010:=[[16.237350545,-0.97869221,0.000576295],[0.999325889,-0.000359757,-0.00001535,-0.036710189],[0,0,0,0],[9E+09,9E+09,9E+09,9E+09,9E+09,9E+09]];
    CONST robtarget H3_1020:=[[19.080365063,-1.194899342,0.000763309],[0.999231859,-0.000454435,-0.000019435,-0.039185262],[0,0,0,0],[9E+09,9E+09,9E+09,9E+09,9E+09,9E+09]];
    CONST robtarget H3_1030:=[[21.249580962,-1.369506366,0.000941132],[0.999154087,-0.000529975,-0.000022818,-0.041119685],[0,0,0,0],[9E+09,9E+09,9E+09,9E+09,9E+09,9E+09]];
    CONST robtarget H3_1040:=[[23.448919217,-1.55526136,0.001155655],[0.999069644,-0.000607444,-0.000026543,-0.043121662],[0,0,0,0],[9E+09,9E+09,9E+09,9E+09,9E+09,9E+09]];
    CONST robtarget H3_1050:=[[27.129145775,-1.886298673,0.001601515],[0.998914071,-0.000737564,-0.000034275,-0.046584695],[0,0,0,0],[9E+09,9E+09,9E+09,9E+09,9E+09,9E+09]];
    CONST robtarget H3_1060:=[[29.99377483,-2.162142024,0.002038094],[0.998779163,-0.000845216,-0.000041759,-0.049390963],[0,0,0,0],[9E+09,9E+09,9E+09,9E+09,9E+09,9E+09]];
    CONST robtarget H3_1070:=[[34.885007358,-2.671653849,0.003002608],[0.998518585,-0.001043716,-0.000057,-0.054401686],[0,0,0,0],[9E+09,9E+09,9E+09,9E+09,9E+09,9E+09]];
    CONST robtarget H3_1080:=[[38.06753586,-3.030407586,0.003803123],[0.998326766,-0.001183656,-0.00006842,-0.057812307],[0,0,0,0],[9E+09,9E+09,9E+09,9E+09,9E+09,9E+09]];
    CONST robtarget H3_1090:=[[42.158116182,-3.524678994,0.005069519],[0.998050038,-0.001376056,-0.000085982,-0.06240369],[0,0,0,0],[9E+09,9E+09,9E+09,9E+09,9E+09,9E+09]];
    CONST robtarget H3_1100:=[[46.372468134,-4.07497443,0.006705876],[0.997725447,-0.001589945,-0.000107567,-0.067389864],[0,0,0,0],[9E+09,9E+09,9E+09,9E+09,9E+09,9E+09]];
    CONST robtarget H3_1110:=[[50.889962806,-4.713759303,0.008898672],[0.997330063,-0.001830876,-0.00013356,-0.073002576],[0,0,0,0],[9E+09,9E+09,9E+09,9E+09,9E+09,9E+09]];
    CONST robtarget H3_1120:=[[54.403390319,-5.247340447,0.010961126],[0.996981235,-0.001997848,-0.000160395,-0.077617005],[0,0,0,0],[9E+09,9E+09,9E+09,9E+09,9E+09,9E+09]];
    CONST robtarget H3_1130:=[[58.252038841,-5.871274564,0.013655874],[0.996548524,-0.002188456,-0.000197025,-0.082983197],[0,0,0,0],[9E+09,9E+09,9E+09,9E+09,9E+09,9E+09]];
    CONST robtarget H3_1140:=[[61.998527955,-6.52080297,0.016796173],[0.996071361,-0.00242225,-0.000236115,-0.088520737],[0,0,0,0],[9E+09,9E+09,9E+09,9E+09,9E+09,9E+09]];
    CONST robtarget H3_1150:=[[66.702193711,-7.399174169,0.021586202],[0.995385782,-0.00281049,-0.000285848,-0.095912277],[0,0,0,0],[9E+09,9E+09,9E+09,9E+09,9E+09,9E+09]];
    CONST robtarget H3_1160:=[[71.172060031,-8.303218002,0.027150401],[0.994635667,-0.003215752,-0.000337737,-0.103389725],[0,0,0,0],[9E+09,9E+09,9E+09,9E+09,9E+09,9E+09]];
    CONST robtarget H3_1170:=[[75.170535937,-9.17311146,0.033086806],[0.993868469,-0.003555064,-0.000395345,-0.110510956],[0,0,0,0],[9E+09,9E+09,9E+09,9E+09,9E+09,9E+09]];
    CONST robtarget H3_1180:=[[79.714378854,-10.237903562,0.04114753],[0.992852446,-0.003954097,-0.000477743,-0.119281841],[0,0,0,0],[9E+09,9E+09,9E+09,9E+09,9E+09,9E+09]];
    CONST robtarget H3_1190:=[[84.250420586,-11.389189518,0.050861466],[0.991666146,-0.004402461,-0.000572198,-0.1287577],[0,0,0,0],[9E+09,9E+09,9E+09,9E+09,9E+09,9E+09]];
    CONST robtarget H3_1200:=[[87.295109808,-12.215539212,0.058465012],[0.990757204,-0.004716625,-0.000645341,-0.135563638],[0,-1,0,0],[9E+09,9E+09,9E+09,9E+09,9E+09,9E+09]];
    CONST robtarget H3_1210:=[[91.414646997,-13.408207067,0.07037304],[0.989352815,-0.005167361,-0.000759633,-0.145443214],[0,-1,0,0],[9E+09,9E+09,9E+09,9E+09,9E+09,9E+09]];
    CONST robtarget H3_1220:=[[95.083542244,-14.549107891,0.082795291],[0.987878219,-0.005595904,-0.0008788,-0.155127487],[0,-1,0,0],[9E+09,9E+09,9E+09,9E+09,9E+09,9E+09]];
    CONST robtarget H3_1230:=[[98.880640635,-15.554633524,0.094581611],[0.99533399,-0.005991345,-0.000586602,-0.096301652],[0,-1,0,0],[9E+09,9E+09,9E+09,9E+09,9E+09,9E+09]];
    CONST robtarget H3_1240:=[[101.932187811,-16.070429391,0.10092624],[0.997781213,-0.006231275,-0.000414484,-0.066284621],[0,-1,0,0],[9E+09,9E+09,9E+09,9E+09,9E+09,9E+09]];
    CONST robtarget H3_1250:=[[105.854430702,-16.323096922,0.104111101],[0.999949865,-0.006350246,0.000048929,0.007742073],[0,-1,0,0],[9E+09,9E+09,9E+09,9E+09,9E+09,9E+09]];
    CONST robtarget H3_1260:=[[109.554313283,-15.960126979,0.099551535],[0.996092697,-0.00618604,0.000547043,0.088095249],[0,-1,0,0],[9E+09,9E+09,9E+09,9E+09,9E+09,9E+09]];
    CONST robtarget H3_1270:=[[113.245241157,-15.019508805,0.088208487],[0.987255244,-0.005771458,0.000929455,0.159037444],[0,-1,0,0],[9E+09,9E+09,9E+09,9E+09,9E+09,9E+09]];
    CONST robtarget H3_1280:=[[116.937211089,-13.519558577,0.071540692],[0.974807538,-0.005133355,0.001174252,0.222985502],[0,-1,0,0],[9E+09,9E+09,9E+09,9E+09,9E+09,9E+09]];
    CONST robtarget H3_1290:=[[120.427465127,-11.571337264,0.052491566],[0.960131277,-0.004331141,0.001260991,0.279513117],[0,-1,0,0],[9E+09,9E+09,9E+09,9E+09,9E+09,9E+09]];
    CONST robtarget H3_1300:=[[123.123512589,-9.679394946,0.036812332],[0.94661793,-0.003574847,0.00121733,0.32233559],[0,-1,0,0],[9E+09,9E+09,9E+09,9E+09,9E+09,9E+09]];
    CONST robtarget H3_1310:=[[125.866551762,-7.350273772,0.021330066],[0.930282222,-0.002669925,0.001053548,0.366833407],[0,-1,1,0],[9E+09,9E+09,9E+09,9E+09,9E+09,9E+09]];
    CONST robtarget H3_1320:=[[129.026066646,-4.02108806,0.006535786],[0.906370763,-0.00142529,0.000664272,0.422480257],[0,-1,1,0],[9E+09,9E+09,9E+09,9E+09,9E+09,9E+09]];
    CONST robtarget H3_1330:=[[131.165000908,-1.210355402,0.00078135],[0.884853428,-0.000419083,0.000220295,0.465869281],[0,-1,1,0],[9E+09,9E+09,9E+09,9E+09,9E+09,9E+09]];
    CONST robtarget H3_1340:=[[133.014189103,1.800951078,0.001480064],[0.859697677,0.000607023,-0.000360685,0.510802707],[0,-1,1,0],[9E+09,9E+09,9E+09,9E+09,9E+09,9E+09]];
    CONST robtarget H3_1350:=[[134.990433074,6.195726668,0.015271793],[0.817495748,0.001989529,-0.001401709,0.575929492],[0,-1,1,0],[9E+09,9E+09,9E+09,9E+09,9E+09,9E+09]];
    CONST robtarget H3_1360:=[[136.274862691,11.211793283,0.049610084],[0.760051237,0.003354173,-0.002867841,0.649848168],[0,-1,1,0],[9E+09,9E+09,9E+09,9E+09,9E+09,9E+09]];
    CONST robtarget H3_1370:=[[136.616894726,15.260226586,0.091832553],[0.712125078,0.004285879,-0.004222843,0.702026831],[0,-1,1,0],[9E+09,9E+09,9E+09,9E+09,9E+09,9E+09]];
    CONST robtarget H3_1380:=[[136.385023396,19.492501763,0.149881342],[0.662753422,0.00510269,-0.005765174,0.748798121],[0,0,0,0],[9E+09,9E+09,9E+09,9E+09,9E+09,9E+09]];
    CONST robtarget H3_1390:=[[135.657343506,23.445416095,0.21698408],[0.616994877,0.005723202,-0.007299371,0.786912502],[0,0,0,0],[9E+09,9E+09,9E+09,9E+09,9E+09,9E+09]];
    CONST robtarget H3_1400:=[[134.713277934,26.633299392,0.280196422],[0.579662657,0.006116242,-0.008597148,0.814788245],[0,0,0,0],[9E+09,9E+09,9E+09,9E+09,9E+09,9E+09]];
    CONST robtarget H3_1410:=[[133.875255901,28.818612544,0.328232705],[0.553346691,0.006323441,-0.009517764,0.832872659],[0,0,0,0],[9E+09,9E+09,9E+09,9E+09,9E+09,9E+09]];
    CONST robtarget H3_1420:=[[132.488926196,31.718406519,0.384252259],[0.516789753,0.004431617,-0.00734104,0.856069402],[0,0,0,0],[9E+09,9E+09,9E+09,9E+09,9E+09,9E+09]];
    CONST robtarget H3_1430:=[[130.645502637,34.833382961,0.443977482],[0.473462633,0.005017788,-0.009335119,0.880750142],[0,0,0,0],[9E+09,9E+09,9E+09,9E+09,9E+09,9E+09]];
    CONST robtarget H3_1440:=[[128.697908722,37.514209587,0.505514576],[0.435222218,0.005378539,-0.011123384,0.900238281],[0,0,0,0],[9E+09,9E+09,9E+09,9E+09,9E+09,9E+09]];
    CONST robtarget H3_1450:=[[126.205325246,40.39502875,0.582189522],[0.397908517,0.005672774,-0.013077934,0.917314341],[0,0,0,0],[9E+09,9E+09,9E+09,9E+09,9E+09,9E+09]];
    CONST robtarget H3_1460:=[[123.117193691,43.472311235,0.676242385],[0.368384667,0.006003936,-0.015154721,0.92953054],[0,0,0,0],[9E+09,9E+09,9E+09,9E+09,9E+09,9E+09]];
    CONST robtarget H3_1470:=[[120.397745774,45.950665657,0.761205745],[0.35620842,0.006399872,-0.016785062,0.934233838],[0,0,0,0],[9E+09,9E+09,9E+09,9E+09,9E+09,9E+09]];
    CONST robtarget H3_1480:=[[116.172358309,48.52414618,0.858180701],[0.260285431,0.005128612,-0.01902136,0.96533071],[0,0,0,0],[9E+09,9E+09,9E+09,9E+09,9E+09,9E+09]];
    CONST robtarget H3_1490:=[[112.93760178,50.34439616,0.932194678],[0.247224462,0.005176493,-0.020286333,0.968732024],[0,0,0,0],[9E+09,9E+09,9E+09,9E+09,9E+09,9E+09]];
    CONST robtarget H3_1500:=[[110.314832364,51.741903709,0.99208104],[0.23785614,0.005207751,-0.021261272,0.971053703],[0,0,0,0],[9E+09,9E+09,9E+09,9E+09,9E+09,9E+09]];
    CONST robtarget H3_10:=[[-112.784408444,-90.444655227,3.125700141],[0.728778058,-0.02484643,0.023316465,0.683901704],[-1,1,-1,0],[9E+09,9E+09,9E+09,9E+09,9E+09,9E+09]];
    CONST robtarget Target_30:=[[17.179545923,-96.959043551,-138.498614445],[0.994633513,0.088387154,0.004759991,-0.05356518],[0,-1,-1,0],[9E+09,9E+09,9E+09,9E+09,9E+09,9E+09]];
    CONST robtarget Target_40:=[[0,0,0],[1,0,0,0],[-1,0,-1,0],[9E+09,9E+09,9E+09,9E+09,9E+09,9E+09]];
    CONST robtarget Target_50:=[[113.316,-96.223,3.532],[1,0,0,0],[0,-2,1,0],[9E+09,9E+09,9E+09,9E+09,9E+09,9E+09]];
    CONST robtarget Target_60:=[[-113.316,-96.222,3.532],[1,0,0,0],[-1,1,-2,0],[9E+09,9E+09,9E+09,9E+09,9E+09,9E+09]];
    CONST robtarget Target_70:=[[200.000039746,-583.667267737,-122.361700735],[0.611889319,0.354388798,-0.354388817,0.611889375],[0,-1,1,0],[9E+09,9E+09,9E+09,9E+09,9E+09,9E+09]];
    CONST robtarget Target_80:=[[-196.999956085,-586.860472861,-123.704824659],[-0.000000016,0.000000048,-0.46295826,0.886380082],[-1,-2,-1,1],[9E+09,9E+09,9E+09,9E+09,9E+09,9E+09]];
    CONST robtarget Target_90:=[[200.000038095,-605.033912372,-79.126916289],[0.74121585,0.065867423,-0.059130623,0.665405227],[0,-2,-2,0],[9E+09,9E+09,9E+09,9E+09,9E+09,9E+09]];
    CONST robtarget Target_100:=[[200.000037341,-599.797758419,-71.91965899],[0.74121585,0.065867423,-0.059130623,0.665405227],[0,-2,-2,0],[9E+09,9E+09,9E+09,9E+09,9E+09,9E+09]];
    CONST robtarget Target_110:=[[200.000036814,-596.23450264,-66.801123237],[0.74121585,0.065867423,-0.059130623,0.665405227],[0,-2,-2,0],[9E+09,9E+09,9E+09,9E+09,9E+09,9E+09]];
    CONST robtarget Target_120:=[[200.000036076,-591.242712572,-59.63053052],[0.74121585,0.065867423,-0.059130623,0.665405227],[0,-2,-2,0],[9E+09,9E+09,9E+09,9E+09,9E+09,9E+09]];
    CONST robtarget Target_130:=[[200.000035405,-586.707439401,-53.115713925],[0.74121585,0.065867423,-0.059130623,0.665405227],[0,-2,-2,0],[9E+09,9E+09,9E+09,9E+09,9E+09,9E+09]];
    CONST robtarget Target_140:=[[200.000033768,-575.643570608,-37.222718445],[0.74121585,0.065867423,-0.059130623,0.665405227],[0,-2,-2,0],[9E+09,9E+09,9E+09,9E+09,9E+09,9E+09]];
    CONST robtarget Target_150:=[[200.000032049,-564.034394952,-20.511748378],[0.74121585,0.065867423,-0.059130623,0.665405227],[0,-2,-2,0],[9E+09,9E+09,9E+09,9E+09,9E+09,9E+09]];
    CONST robtarget Target_160:=[[200.000030036,-551.456474976,-0.112153845],[0.74121585,0.065867423,-0.059130623,0.665405227],[0,-2,-2,0],[9E+09,9E+09,9E+09,9E+09,9E+09,9E+09]];
    CONST robtarget Target_170:=[[200.000028223,-540.515811383,18.595217139],[0.74121585,0.065867423,-0.059130623,0.665405227],[0,-2,-2,0],[9E+09,9E+09,9E+09,9E+09,9E+09,9E+09]];
    CONST robtarget Target_180:=[[200.000025867,-526.47340748,43.046542514],[0.74121585,0.065867423,-0.059130623,0.665405227],[0,-2,-2,0],[9E+09,9E+09,9E+09,9E+09,9E+09,9E+09]];
    CONST robtarget Target_190:=[[200.000023154,-510.388336841,71.282365427],[0.74121585,0.065867423,-0.059130623,0.665405227],[0,-2,-2,0],[9E+09,9E+09,9E+09,9E+09,9E+09,9E+09]];
    CONST robtarget Target_200:=[[200.000021531,-500.758829808,88.15579517],[0.74121585,0.065867423,-0.059130623,0.665405227],[0,-2,-2,0],[9E+09,9E+09,9E+09,9E+09,9E+09,9E+09]];
    CONST robtarget Target_210:=[[200.000020096,-492.158408599,103.010121308],[0.74121585,0.065867423,-0.059130623,0.665405227],[0,-2,-2,0],[9E+09,9E+09,9E+09,9E+09,9E+09,9E+09]];
    CONST robtarget Target_220:=[[200.000019078,-485.398457656,112.996628818],[0.74121585,0.065867423,-0.059130623,0.665405227],[0,-2,-2,0],[9E+09,9E+09,9E+09,9E+09,9E+09,9E+09]];
    CONST robtarget Target_230:=[[200.000017806,-475.074404862,123.906076738],[0.74121585,0.065867423,-0.059130623,0.665405227],[0,-2,-2,0],[9E+09,9E+09,9E+09,9E+09,9E+09,9E+09]];
    CONST robtarget Target_240:=[[200.000016891,-466.319538356,130.639381534],[0.74121585,0.065867423,-0.059130623,0.665405227],[0,-2,-2,0],[9E+09,9E+09,9E+09,9E+09,9E+09,9E+09]];
    CONST robtarget Target_250:=[[200.000016094,-457.573199438,135.565869991],[0.74121585,0.065867423,-0.059130623,0.665405227],[0,-2,-2,0],[9E+09,9E+09,9E+09,9E+09,9E+09,9E+09]];
    CONST robtarget Target_260:=[[200.000014873,-441.549440966,140.932523924],[0.74121585,0.065867423,-0.059130623,0.665405227],[0,-2,-2,0],[9E+09,9E+09,9E+09,9E+09,9E+09,9E+09]];
    CONST robtarget Target_270:=[[200.000013685,-421.65690905,142.538450129],[0.74121585,0.065867423,-0.059130623,0.665405227],[0,-2,-2,0],[9E+09,9E+09,9E+09,9E+09,9E+09,9E+09]];
    CONST robtarget Target_280:=[[200.000012906,-404.988152487,140.561770932],[0.74121585,0.065867423,-0.059130623,0.665405227],[0,-2,-2,0],[9E+09,9E+09,9E+09,9E+09,9E+09,9E+09]];
    CONST robtarget Target_290:=[[200.00001212,-383.148107462,134.358747612],[0.74121585,0.065867423,-0.059130623,0.665405227],[0,-2,-2,0],[9E+09,9E+09,9E+09,9E+09,9E+09,9E+09]];
    CONST robtarget Target_300:=[[200.000011606,-361.13927251,123.844938406],[0.74121585,0.065867423,-0.059130623,0.665405227],[0,-2,-2,0],[9E+09,9E+09,9E+09,9E+09,9E+09,9E+09]];
    CONST robtarget Target_310:=[[200.00001144,-349.585673011,116.724675515],[0.74121585,0.065867423,-0.059130623,0.665405227],[0,-2,-2,0],[9E+09,9E+09,9E+09,9E+09,9E+09,9E+09]];
    CONST robtarget Target_320:=[[200.000011216,-335.072217299,108.01950531],[0.74121585,0.065867423,-0.059130623,0.665405227],[0,-2,-2,0],[9E+09,9E+09,9E+09,9E+09,9E+09,9E+09]];
    CONST robtarget Target_330:=[[198.432010925,-317.680730828,97.942335201],[0.74121585,0.065867423,-0.059130623,0.665405227],[0,-2,1,0],[9E+09,9E+09,9E+09,9E+09,9E+09,9E+09]];
    CONST robtarget Target_340:=[[196.383010812,-301.092518704,85.799144885],[0.74121585,0.065867423,-0.059130623,0.665405227],[0,0,0,0],[9E+09,9E+09,9E+09,9E+09,9E+09,9E+09]];
    CONST robtarget Target_350:=[[195.032010672,-289.479328545,78.238488963],[0.74121585,0.065867423,-0.059130623,0.665405227],[0,0,0,0],[9E+09,9E+09,9E+09,9E+09,9E+09,9E+09]];
    CONST robtarget Target_360:=[[193.373010423,-274.622607482,69.630369341],[0.74121585,0.065867423,-0.059130623,0.665405227],[0,0,0,0],[9E+09,9E+09,9E+09,9E+09,9E+09,9E+09]];
    CONST robtarget Target_370:=[[191.385010027,-256.131260333,60.23584072],[0.74121585,0.065867423,-0.059130623,0.665405227],[0,0,0,0],[9E+09,9E+09,9E+09,9E+09,9E+09,9E+09]];
    CONST robtarget Target_380:=[[189.630009601,-239.29713476,52.697165987],[0.74121585,0.065867423,-0.059130623,0.665405227],[0,0,0,0],[9E+09,9E+09,9E+09,9E+09,9E+09,9E+09]];
    CONST robtarget Target_390:=[[188.113009182,-224.427302694,46.698244164],[0.74121585,0.065867423,-0.059130623,0.665405227],[0,0,0,0],[9E+09,9E+09,9E+09,9E+09,9E+09,9E+09]];
    CONST robtarget Target_400:=[[186.583008717,-209.183114105,41.093511625],[0.74121585,0.065867423,-0.059130623,0.665405227],[0,0,0,0],[9E+09,9E+09,9E+09,9E+09,9E+09,9E+09]];
    CONST robtarget Target_410:=[[185.120008236,-194.401777981,36.115990053],[0.74121585,0.065867423,-0.059130623,0.665405227],[0,0,0,0],[9E+09,9E+09,9E+09,9E+09,9E+09,9E+09]];
    CONST robtarget Target_420:=[[183.108007522,-173.780265101,29.824713104],[0.74121585,0.065867423,-0.059130623,0.665405227],[0,0,0,0],[9E+09,9E+09,9E+09,9E+09,9E+09,9E+09]];
    CONST robtarget Target_430:=[[181.554006934,-157.66004483,25.369468488],[0.74121585,0.065867423,-0.059130623,0.665405227],[0,0,0,0],[9E+09,9E+09,9E+09,9E+09,9E+09,9E+09]];
    CONST robtarget Target_440:=[[180.560006543,-147.26771592,22.690019281],[0.74121585,0.065867423,-0.059130623,0.665405227],[0,0,0,0],[9E+09,9E+09,9E+09,9E+09,9E+09,9E+09]];
    CONST robtarget Target_450:=[[179.427005924,-133.765048124,20.891842988],[0.74121585,0.065867423,-0.059130623,0.665405227],[0,0,0,0],[9E+09,9E+09,9E+09,9E+09,9E+09,9E+09]];
    CONST robtarget Target_460:=[[178.08000517,-117.261577837,18.675258573],[0.74121585,0.065867423,-0.059130623,0.665405227],[0,0,0,0],[9E+09,9E+09,9E+09,9E+09,9E+09,9E+09]];
    CONST robtarget Target_470:=[[176.463004424,-99.033785288,14.886091335],[0.74121585,0.065867423,-0.059130623,0.665405227],[0,0,0,0],[9E+09,9E+09,9E+09,9E+09,9E+09,9E+09]];
    CONST robtarget Target_480:=[[174.8810038,-82.430011441,10.578426994],[0.74121585,0.065867423,-0.059130623,0.665405227],[0,0,0,0],[9E+09,9E+09,9E+09,9E+09,9E+09,9E+09]];
    CONST robtarget Target_490:=[[173.828003427,-71.922545484,7.528474801],[0.74121585,0.065867423,-0.059130623,0.665405227],[0,0,0,0],[9E+09,9E+09,9E+09,9E+09,9E+09,9E+09]];
    CONST robtarget Target_500:=[[172.872003111,-62.730778122,4.688813349],[0.74121585,0.065867423,-0.059130623,0.665405227],[0,0,0,0],[9E+09,9E+09,9E+09,9E+09,9E+09,9E+09]];
    CONST robtarget Target_510:=[[171.784002774,-52.612204417,1.399535397],[0.74121585,0.065867423,-0.059130623,0.665405227],[0,0,0,0],[9E+09,9E+09,9E+09,9E+09,9E+09,9E+09]];
    CONST robtarget Target_520:=[[170.495002402,-41.08888517,-2.529053861],[0.74121585,0.065867423,-0.059130623,0.665405227],[0,0,0,0],[9E+09,9E+09,9E+09,9E+09,9E+09,9E+09]];
    CONST robtarget Target_530:=[[169.71700219,-34.358373258,-4.905463143],[0.74121585,0.065867423,-0.059130623,0.665405227],[0,0,0,0],[9E+09,9E+09,9E+09,9E+09,9E+09,9E+09]];
    CONST robtarget Target_540:=[[168.321001831,-22.673463893,-9.157628724],[0.74121585,0.065867423,-0.059130623,0.665405227],[0,0,0,0],[9E+09,9E+09,9E+09,9E+09,9E+09,9E+09]];
    CONST robtarget Target_550:=[[166.063001299,-4.784304032,-15.950577941],[0.74121585,0.065867423,-0.059130623,0.665405227],[0,0,0,0],[9E+09,9E+09,9E+09,9E+09,9E+09,9E+09]];
    CONST robtarget Target_560:=[[163.967000851,10.805304455,-22.111110006],[0.74121585,0.065867423,-0.059130623,0.665405227],[0,0,0,0],[9E+09,9E+09,9E+09,9E+09,9E+09,9E+09]];
    CONST robtarget Target_570:=[[161.930000452,25.076079972,-27.924763722],[0.74121585,0.065867423,-0.059130623,0.665405227],[0,0,0,0],[9E+09,9E+09,9E+09,9E+09,9E+09,9E+09]];
    CONST robtarget Target_580:=[[160.246000004,37.228513312,-31.208310037],[0.74121585,0.065867423,-0.059130623,0.665405227],[0,0,0,0],[9E+09,9E+09,9E+09,9E+09,9E+09,9E+09]];
    CONST robtarget Target_590:=[[157.368999383,53.207612143,-35.034583547],[0.74121585,0.065867423,-0.059130623,0.665405227],[0,0,0,0],[9E+09,9E+09,9E+09,9E+09,9E+09,9E+09]];
    CONST robtarget Target_600:=[[152.833999153,63.224460321,-39.888314329],[0.74121585,0.065867423,-0.059130623,0.665405227],[0,1,-1,0],[9E+09,9E+09,9E+09,9E+09,9E+09,9E+09]];
    CONST robtarget Target_610:=[[143.451998924,74.60520066,-45.890539419],[0.74121585,0.065867423,-0.059130623,0.665405227],[0,1,-1,0],[9E+09,9E+09,9E+09,9E+09,9E+09,9E+09]];
    CONST robtarget Target_620:=[[127.744998706,86.171052049,-52.217207169],[0.74121585,0.065867423,-0.059130623,0.665405227],[0,1,-1,0],[9E+09,9E+09,9E+09,9E+09,9E+09,9E+09]];
    CONST robtarget Target_630:=[[114.504998568,93.969628986,-56.620032977],[0.74121585,0.065867423,-0.059130623,0.665405227],[0,0,0,0],[9E+09,9E+09,9E+09,9E+09,9E+09,9E+09]];
    CONST robtarget Target_640:=[[100.432998454,100.693026399,-60.499246303],[0.74121585,0.065867423,-0.059130623,0.665405227],[0,0,0,0],[9E+09,9E+09,9E+09,9E+09,9E+09,9E+09]];
    CONST robtarget Target_650:=[[88.039998375,105.546704202,-63.343946958],[0.74121585,0.065867423,-0.059130623,0.665405227],[0,0,0,0],[9E+09,9E+09,9E+09,9E+09,9E+09,9E+09]];
    CONST robtarget Target_660:=[[73.2199983,110.261867792,-66.141331291],[0.74121585,0.065867423,-0.059130623,0.665405227],[0,0,0,0],[9E+09,9E+09,9E+09,9E+09,9E+09,9E+09]];
    CONST robtarget Target_670:=[[59.348998246,113.74321987,-68.227129991],[0.74121585,0.065867423,-0.059130623,0.665405227],[0,0,0,0],[9E+09,9E+09,9E+09,9E+09,9E+09,9E+09]];
    CONST robtarget Target_680:=[[45.087998204,116.489388768,-69.883843966],[0.74121585,0.065867423,-0.059130623,0.665405227],[0,0,0,0],[9E+09,9E+09,9E+09,9E+09,9E+09,9E+09]];
    CONST robtarget Target_690:=[[26.32199811,118.123985983,-69.804361834],[0.74121585,0.065867423,-0.059130623,0.665405227],[0,0,0,0],[9E+09,9E+09,9E+09,9E+09,9E+09,9E+09]];
    CONST robtarget Target_700:=[[6.88699811,118.123984925,-69.804363098],[0.74121585,0.065867423,-0.059130623,0.665405227],[0,0,0,0],[9E+09,9E+09,9E+09,9E+09,9E+09,9E+09]];
    CONST robtarget Target_710:=[[-7.47200189,118.123984143,-69.804364033],[0.74121585,0.065867423,-0.059130623,0.665405227],[0,0,0,0],[9E+09,9E+09,9E+09,9E+09,9E+09,9E+09]];
    CONST robtarget Target_720:=[[-26.96100189,118.123983081,-69.804365301],[0.74121585,0.065867423,-0.059130623,0.665405227],[0,0,0,0],[9E+09,9E+09,9E+09,9E+09,9E+09,9E+09]];
    CONST robtarget Target_730:=[[-54.063001771,114.855671144,-68.896459732],[0.74121585,0.065867423,-0.059130623,0.665405227],[0,0,0,0],[9E+09,9E+09,9E+09,9E+09,9E+09,9E+09]];
    CONST robtarget Target_740:=[[-83.706001649,107.040700836,-64.226338503],[0.74121585,0.065867423,-0.059130623,0.665405227],[0,0,0,0],[9E+09,9E+09,9E+09,9E+09,9E+09,9E+09]];
    CONST robtarget Target_750:=[[-105.060001512,98.637220578,-59.305056412],[0.74121585,0.065867423,-0.059130623,0.665405227],[0,0,0,0],[9E+09,9E+09,9E+09,9E+09,9E+09,9E+09]];
    CONST robtarget Target_760:=[[-123.430001343,88.893579076,-53.742036327],[0.74121585,0.065867423,-0.059130623,0.665405227],[0,0,0,0],[9E+09,9E+09,9E+09,9E+09,9E+09,9E+09]];
    CONST robtarget Target_770:=[[-145.003001048,73.127504494,-45.093638206],[0.74121585,0.065867423,-0.059130623,0.665405227],[0,0,0,0],[9E+09,9E+09,9E+09,9E+09,9E+09,9E+09]];
    CONST robtarget Target_780:=[[-156.960000648,54.425636516,-35.584435733],[0.74121585,0.065867423,-0.059130623,0.665405227],[0,0,0,0],[9E+09,9E+09,9E+09,9E+09,9E+09,9E+09]];
    CONST robtarget Target_790:=[[-161.502999643,28.063606993,-28.972390166],[0.74121585,0.065867423,-0.059130623,0.665405227],[0,0,0,0],[9E+09,9E+09,9E+09,9E+09,9E+09,9E+09]];
    CONST robtarget Target_800:=[[-165.115998909,2.37289356,-18.752432015],[0.74121585,0.065867423,-0.059130623,0.665405227],[0,0,0,0],[9E+09,9E+09,9E+09,9E+09,9E+09,9E+09]];
    CONST robtarget Target_810:=[[-167.676998327,-17.45497123,-11.106987238],[0.74121585,0.065867423,-0.059130623,0.665405227],[0,0,0,0],[9E+09,9E+09,9E+09,9E+09,9E+09,9E+09]];
    CONST robtarget Target_820:=[[-170.8439975,-44.16744886,-1.461199655],[0.74121585,0.065867423,-0.059130623,0.665405227],[0,0,0,0],[9E+09,9E+09,9E+09,9E+09,9E+09,9E+09]];
    CONST robtarget Target_830:=[[-173.278996757,-66.60375128,5.90389161],[0.74121585,0.065867423,-0.059130623,0.665405227],[0,0,0,0],[9E+09,9E+09,9E+09,9E+09,9E+09,9E+09]];
    CONST robtarget Target_840:=[[-175.236996066,-86.077152517,11.582013216],[0.74121585,0.065867423,-0.059130623,0.665405227],[0,0,0,0],[9E+09,9E+09,9E+09,9E+09,9E+09,9E+09]];
    CONST robtarget Target_850:=[[-176.838995414,-103.153494418,15.8395615],[0.74121585,0.065867423,-0.059130623,0.665405227],[0,0,0,0],[9E+09,9E+09,9E+09,9E+09,9E+09,9E+09]];
    CONST robtarget Target_860:=[[-178.752994472,-125.333336707,19.93565093],[0.74121585,0.065867423,-0.059130623,0.665405227],[0,0,0,0],[9E+09,9E+09,9E+09,9E+09,9E+09,9E+09]];
    CONST robtarget Target_870:=[[-181.657993025,-158.742566403,25.65605236],[0.74121585,0.065867423,-0.059130623,0.665405227],[0,0,0,0],[9E+09,9E+09,9E+09,9E+09,9E+09,9E+09]];
    CONST robtarget Target_880:=[[-184.1539921,-184.545505806,33.020475202],[0.74121585,0.065867423,-0.059130623,0.665405227],[0,0,0,0],[9E+09,9E+09,9E+09,9E+09,9E+09,9E+09]];
    CONST robtarget Target_890:=[[-186.238991393,-205.726951642,39.891094041],[0.74121585,0.065867423,-0.059130623,0.665405227],[0,0,0,0],[9E+09,9E+09,9E+09,9E+09,9E+09,9E+09]];
    CONST robtarget Target_900:=[[-188.27899077,-226.074553398,47.335744289],[0.74121585,0.065867423,-0.059130623,0.665405227],[0,0,0,0],[9E+09,9E+09,9E+09,9E+09,9E+09,9E+09]];
    CONST robtarget Target_910:=[[-190.285990232,-245.641938494,55.438283562],[0.74121585,0.065867423,-0.059130623,0.665405227],[0,0,0,0],[9E+09,9E+09,9E+09,9E+09,9E+09,9E+09]];
    CONST robtarget Target_920:=[[-193.279989593,-273.769470609,69.166518189],[0.74121585,0.065867423,-0.059130623,0.665405227],[0,0,0,0],[9E+09,9E+09,9E+09,9E+09,9E+09,9E+09]];
    CONST robtarget Target_930:=[[-195.927989228,-297.239632492,83.198777027],[0.74121585,0.065867423,-0.059130623,0.665405227],[0,0,0,0],[9E+09,9E+09,9E+09,9E+09,9E+09,9E+09]];
    CONST robtarget Target_940:=[[-198.501989072,-318.220551425,98.352552054],[0.74121585,0.065867423,-0.059130623,0.665405227],[0,0,0,0],[9E+09,9E+09,9E+09,9E+09,9E+09,9E+09]];
    CONST robtarget Target_950:=[[-199.999988537,-351.176404449,117.704504979],[0.74121585,0.065867423,-0.059130623,0.665405227],[0,0,0,0],[9E+09,9E+09,9E+09,9E+09,9E+09,9E+09]];
    CONST robtarget Target_960:=[[-199.999987625,-390.990070206,137.007412947],[0.74121585,0.065867423,-0.059130623,0.665405227],[0,0,0,0],[9E+09,9E+09,9E+09,9E+09,9E+09,9E+09]];
    CONST robtarget Target_970:=[[-199.999987132,-404.07990395,140.380058282],[0.74121585,0.065867423,-0.059130623,0.665405227],[0,0,0,0],[9E+09,9E+09,9E+09,9E+09,9E+09,9E+09]];
    CONST robtarget Target_980:=[[-199.999986307,-421.808254426,142.543824994],[0.74121585,0.065867423,-0.059130623,0.665405227],[0,0,0,0],[9E+09,9E+09,9E+09,9E+09,9E+09,9E+09]];
    CONST robtarget Target_990:=[[-199.999985356,-438.11570873,141.567948404],[0.74121585,0.065867423,-0.059130623,0.665405227],[0,0,0,0],[9E+09,9E+09,9E+09,9E+09,9E+09,9E+09]];
    CONST robtarget Target_1000:=[[-199.999984301,-452.778123634,137.62465166],[0.74121585,0.065867423,-0.059130623,0.665405227],[0,0,0,0],[9E+09,9E+09,9E+09,9E+09,9E+09,9E+09]];
    CONST robtarget Target_1010:=[[-199.999983273,-464.613201597,131.730342915],[0.74121585,0.065867423,-0.059130623,0.665405227],[0,0,0,0],[9E+09,9E+09,9E+09,9E+09,9E+09,9E+09]];
    CONST robtarget Target_1020:=[[-199.999982027,-476.542067165,122.571338642],[0.74121585,0.065867423,-0.059130623,0.665405227],[0,0,0,0],[9E+09,9E+09,9E+09,9E+09,9E+09,9E+09]];
    CONST robtarget Target_1030:=[[-199.999980497,-488.439035849,109.015054006],[0.74121585,0.065867423,-0.059130623,0.665405227],[0,0,0,0],[9E+09,9E+09,9E+09,9E+09,9E+09,9E+09]];
    CONST robtarget Target_1040:=[[-199.999978679,-499.505372517,90.340029247],[0.74121585,0.065867423,-0.059130623,0.665405227],[0,0,0,0],[9E+09,9E+09,9E+09,9E+09,9E+09,9E+09]];
    CONST robtarget Target_1050:=[[-199.999976225,-514.06752532,64.820312051],[0.74121585,0.065867423,-0.059130623,0.665405227],[0,0,0,0],[9E+09,9E+09,9E+09,9E+09,9E+09,9E+09]];
    CONST robtarget Target_1060:=[[-199.999973189,-532.082579913,33.242800354],[0.74121585,0.065867423,-0.059130623,0.665405227],[0,0,0,0],[9E+09,9E+09,9E+09,9E+09,9E+09,9E+09]];
    CONST robtarget Target_1070:=[[-199.999971085,-544.675153904,11.433532363],[0.74121585,0.065867423,-0.059130623,0.665405227],[0,0,0,0],[9E+09,9E+09,9E+09,9E+09,9E+09,9E+09]];
    CONST robtarget Target_1080:=[[-199.99996863,-559.686163155,-13.718573776],[0.74121585,0.065867423,-0.059130623,0.665405227],[0,0,0,0],[9E+09,9E+09,9E+09,9E+09,9E+09,9E+09]];
    CONST robtarget Target_1090:=[[-199.999965986,-577.304829097,-39.609073162],[0.74121585,0.065867423,-0.059130623,0.665405227],[0,0,0,0],[9E+09,9E+09,9E+09,9E+09,9E+09,9E+09]];
    CONST robtarget Target_1100:=[[-199.999963644,-593.134249496,-62.347674962],[0.74121585,0.065867423,-0.059130623,0.665405227],[0,0,0,0],[9E+09,9E+09,9E+09,9E+09,9E+09,9E+09]];
    CONST robtarget Target_1110:=[[-199.999961428,-608.495829169,-83.546654064],[0.74121585,0.065867423,-0.059130623,0.665405227],[0,0,0,0],[9E+09,9E+09,9E+09,9E+09,9E+09,9E+09]];
    CONST robtarget Target_1140:=[[-192.856957763,-640.588033516,-113.011360558],[0.954126456,-0.299403916,-0.000000039,0.000000016],[-1,1,-2,0],[9E+09,9E+09,9E+09,9E+09,9E+09,9E+09]];
    CONST robtarget Target_1150:=[[-183.370957763,-640.588033,-113.011359941],[0.954126456,-0.299403916,-0.000000039,0.000000016],[-1,1,-2,0],[9E+09,9E+09,9E+09,9E+09,9E+09,9E+09]];
    CONST robtarget Target_1160:=[[-170.688957763,-640.588032309,-113.011359115],[0.954126456,-0.299403916,-0.000000039,0.000000016],[-1,1,-2,0],[9E+09,9E+09,9E+09,9E+09,9E+09,9E+09]];
    CONST robtarget Target_1170:=[[-158.166957763,-640.588031627,-113.011358301],[0.954126456,-0.299403916,-0.000000039,0.000000016],[-1,1,-2,0],[9E+09,9E+09,9E+09,9E+09,9E+09,9E+09]];
    CONST robtarget Target_1180:=[[-142.511957763,-640.588030775,-113.011357282],[0.954126456,-0.299403916,-0.000000039,0.000000016],[-1,1,-2,0],[9E+09,9E+09,9E+09,9E+09,9E+09,9E+09]];
    CONST robtarget Target_1190:=[[-128.099957763,-640.58802999,-113.011356344],[0.954126456,-0.299403916,-0.000000039,0.000000016],[-1,1,-2,0],[9E+09,9E+09,9E+09,9E+09,9E+09,9E+09]];
    CONST robtarget Target_1200:=[[-99.370957763,-640.588028425,-113.011354474],[0.954126456,-0.299403916,-0.000000039,0.000000016],[-1,1,-2,0],[9E+09,9E+09,9E+09,9E+09,9E+09,9E+09]];
    CONST robtarget Target_1210:=[[-75.151957763,-640.588027107,-113.011352898],[0.954126456,-0.299403916,-0.000000039,0.000000016],[-1,1,-2,0],[9E+09,9E+09,9E+09,9E+09,9E+09,9E+09]];
    CONST robtarget Target_1220:=[[-56.803957763,-640.588026108,-113.011351704],[0.954126456,-0.299403916,-0.000000039,0.000000016],[-1,1,-2,0],[9E+09,9E+09,9E+09,9E+09,9E+09,9E+09]];
    CONST robtarget Target_1230:=[[-31.012957763,-640.588024703,-113.011350026],[0.954126456,-0.299403916,-0.000000039,0.000000016],[-1,1,-2,0],[9E+09,9E+09,9E+09,9E+09,9E+09,9E+09]];
    CONST robtarget Target_1240:=[[7.645042237,-640.588022598,-113.01134751],[0.954126456,-0.299403916,-0.000000039,0.000000016],[0,-2,1,0],[9E+09,9E+09,9E+09,9E+09,9E+09,9E+09]];
    CONST robtarget Target_1250:=[[30.058042237,-640.588021378,-113.011346052],[0.954126456,-0.299403916,-0.000000039,0.000000016],[0,-2,1,0],[9E+09,9E+09,9E+09,9E+09,9E+09,9E+09]];
    CONST robtarget Target_1260:=[[59.528042237,-640.588019773,-113.011344134],[0.954126456,-0.299403916,-0.000000039,0.000000016],[0,-2,1,0],[9E+09,9E+09,9E+09,9E+09,9E+09,9E+09]];
    CONST robtarget Target_1270:=[[91.830042237,-640.588018014,-113.011342032],[0.954126456,-0.299403916,-0.000000039,0.000000016],[0,-2,1,0],[9E+09,9E+09,9E+09,9E+09,9E+09,9E+09]];
    CONST robtarget Target_1280:=[[129.841042237,-640.588015944,-113.011339558],[0.954126456,-0.299403916,-0.000000039,0.000000016],[0,-2,1,0],[9E+09,9E+09,9E+09,9E+09,9E+09,9E+09]];
    CONST robtarget Target_1290:=[[153.028042237,-640.588014681,-113.011338049],[0.954126456,-0.299403916,-0.000000039,0.000000016],[0,-2,1,0],[9E+09,9E+09,9E+09,9E+09,9E+09,9E+09]];
    CONST robtarget Target_1300:=[[175.208042237,-640.588013474,-113.011336606],[0.954126456,-0.299403916,-0.000000039,0.000000016],[0,-2,1,0],[9E+09,9E+09,9E+09,9E+09,9E+09,9E+09]];
    CONST robtarget Target_1310:=[[187.548042237,-640.588012802,-113.011335803],[0.954126456,-0.299403916,-0.000000039,0.000000016],[0,-2,1,0],[9E+09,9E+09,9E+09,9E+09,9E+09,9E+09]];
    CONST robtarget H1_500:=[[-29.461627781,-2.109705055,0.001950535],[0.99880514,-0.000824758,0.000040289,0.04886319],[0,0,0,0],[9E+09,9E+09,9E+09,9E+09,9E+09,9E+09]];
    CONST robtarget H1_510:=[[-19.246148462,-1.207965007,0.000775799],[0.999226044,-0.00047264,0.000019197,0.039333044],[0,0,0,0],[9E+09,9E+09,9E+09,9E+09,9E+09,9E+09]];
    CONST robtarget H1_520:=[[-8.751898287,-0.475188465,0.000289484],[0.999534191,-0.00018602,0.000005268,0.030518288],[0,0,0,0],[9E+09,9E+09,9E+09,9E+09,9E+09,9E+09]];
    CONST robtarget H1_490:=[[-40.43486389,-3.311827817,0.004500669],[0.998171024,-0.001293225,0.000078153,0.060439456],[0,0,0,0],[9E+09,9E+09,9E+09,9E+09,9E+09,9E+09]];
    CONST robtarget H3_30:=[[-113.422700461,-71.025825775,1.937894203],[0.65947976,-0.017804432,0.020281522,0.751237718],[-1,1,-1,0],[9E+09,9E+09,9E+09,9E+09,9E+09,9E+09]];
    CONST robtarget H3_50:=[[-118.579215305,-51.169989193,1.011437027],[0.507056869,-0.009945927,0.016902133,0.861689461],[-1,1,0,0],[9E+09,9E+09,9E+09,9E+09,9E+09,9E+09]];
    CONST robtarget H3_20:=[[-112.64983989,-80.211372212,2.465299429],[0.693331406,-0.021055401,0.021864669,0.719979283],[-1,1,-1,0],[9E+09,9E+09,9E+09,9E+09,9E+09,9E+09]];
    CONST robtarget H3_40:=[[-115.473413237,-60.093263587,1.391452911],[0.617207203,-0.014163786,0.018047982,0.7864661],[-1,1,0,0],[9E+09,9E+09,9E+09,9E+09,9E+09,9E+09]];
    CONST robtarget H3_60:=[[-126.021573344,-42.948884511,0.714225549],[0.247591924,-0.004090617,0.016004784,0.968723569],[-1,1,0,0],[9E+09,9E+09,9E+09,9E+09,9E+09,9E+09]];
    CONST robtarget H3_70:=[[-137.693743744,-43.433535744,0.730333302],[0.254463381,-0.00425073,-0.016152227,-0.96693817],[-1,1,1,0],[9E+09,9E+09,9E+09,9E+09,9E+09,9E+09]];
    CONST robtarget H3_80:=[[-145.82650877,-51.242271974,1.014275784],[0.480909186,-0.009446218,-0.017217468,-0.876550445],[-1,1,1,0],[9E+09,9E+09,9E+09,9E+09,9E+09,9E+09]];
    CONST robtarget Con_100:=[[200.000066114,-463.8631146,49.489390244],[0.61128662,0.355427493,-0.355427462,0.611286581],[0,-1,1,0],[9E+09,9E+09,9E+09,9E+09,9E+09,9E+09]];
    CONST robtarget Con_110:=[[200.000067741,-452.406605334,69.604908922],[0.61147304,0.355106684,-0.355106653,0.611473],[0,-1,1,0],[9E+09,9E+09,9E+09,9E+09,9E+09,9E+09]];
    CONST robtarget Con_520:=[[66.430159526,164.814113195,-78.092499318],[0.138051419,-0.03336851,0.295071588,0.944860363],[0,0,1,1],[9E+09,9E+09,9E+09,9E+09,9E+09,9E+09]];
    CONST robtarget Con_130:=[[200.00007045,-432.237489876,102.643175652],[0.638619039,0.303588137,-0.303588103,0.638619002],[0,-1,1,0],[9E+09,9E+09,9E+09,9E+09,9E+09,9E+09]];
    CONST robtarget Con_140:=[[200.000071909,-415.822319766,118.229718671],[0.673481121,0.215460459,-0.215460421,0.673481089],[0,-1,1,0],[9E+09,9E+09,9E+09,9E+09,9E+09,9E+09]];
    CONST robtarget Con_160:=[[200.000073838,-375.994847219,131.645898369],[0.70694018,0.015349135,-0.015349089,0.706940161],[0,-1,1,0],[9E+09,9E+09,9E+09,9E+09,9E+09,9E+09]];
    CONST robtarget Con_170:=[[200.000074394,-347.015579951,128.549833252],[0.702197427,-0.0831792,0.083179248,0.702197414],[0,0,0,1],[9E+09,9E+09,9E+09,9E+09,9E+09,9E+09]];
    CONST robtarget Con_180:=[[200.000074487,-317.383305715,118.1671017],[0.691355937,-0.148414845,0.148414895,0.691355929],[0,0,0,1],[9E+09,9E+09,9E+09,9E+09,9E+09,9E+09]];
    CONST robtarget Con_190:=[[199.586400944,-273.889876796,93.303181423],[0.640470953,-0.185850679,0.210746467,0.714732405],[0,0,0,1],[9E+09,9E+09,9E+09,9E+09,9E+09,9E+09]];
    CONST robtarget Con_200:=[[196.859402798,-252.311296621,77.708980059],[0.639257735,-0.205635161,0.226008659,0.705679682],[0,0,0,1],[9E+09,9E+09,9E+09,9E+09,9E+09,9E+09]];
    CONST robtarget Con_210:=[[195.324578994,-239.29135035,68.963495382],[0.645969331,-0.18530289,0.207297477,0.710924904],[0,0,0,1],[9E+09,9E+09,9E+09,9E+09,9E+09,9E+09]];
    CONST robtarget Con_220:=[[193.647772138,-224.379858568,60.136109129],[0.651658116,-0.165533269,0.189201442,0.715641845],[0,0,0,1],[9E+09,9E+09,9E+09,9E+09,9E+09,9E+09]];
    CONST robtarget Con_230:=[[192.16221414,-210.693903516,52.92356398],[0.655631095,-0.150002159,0.175029903,0.719035293],[0,0,0,1],[9E+09,9E+09,9E+09,9E+09,9E+09,9E+09]];
    CONST robtarget Con_240:=[[190.302115573,-193.048186799,44.63404443],[0.659567207,-0.132819639,0.159386591,0.722444432],[0,0,0,1],[9E+09,9E+09,9E+09,9E+09,9E+09,9E+09]];
    CONST robtarget Con_250:=[[189.021322288,-180.620397513,39.365478155],[0.661760377,-0.122244682,0.14977687,0.724359255],[0,0,0,1],[9E+09,9E+09,9E+09,9E+09,9E+09,9E+09]];
    CONST robtarget Con_260:=[[187.280613807,-163.422669954,32.727287708],[0.664207361,-0.109323201,0.138055403,0.726510651],[0,0,0,1],[9E+09,9E+09,9E+09,9E+09,9E+09,9E+09]];
    CONST robtarget Con_270:=[[185.520886633,-145.727242462,26.574650477],[0.666194142,-0.097700838,0.127533265,0.728268617],[0,0,0,1],[9E+09,9E+09,9E+09,9E+09,9E+09,9E+09]];
    CONST robtarget Con_280:=[[184.325158093,-133.548844445,22.687091774],[0.667322198,-0.090514346,0.121038095,0.729272251],[0,0,0,1],[9E+09,9E+09,9E+09,9E+09,9E+09,9E+09]];
    CONST robtarget Con_290:=[[182.787616099,-117.727741909,18.009222246],[0.668557914,-0.082012888,0.113366658,0.730378123],[0,0,0,1],[9E+09,9E+09,9E+09,9E+09,9E+09,9E+09]];
    CONST robtarget Con_300:=[[181.48544865,-104.201375352,14.310660091],[0.669445202,-0.075398185,0.107408016,0.731178332],[0,0,0,1],[9E+09,9E+09,9E+09,9E+09,9E+09,9E+09]];
    CONST robtarget Con_310:=[[179.155985689,-77.578305811,9.68158655],[0.67829567,-0.022407117,0.055743166,0.732328891],[0,0,0,1],[9E+09,9E+09,9E+09,9E+09,9E+09,9E+09]];
    CONST robtarget Con_320:=[[177.935201252,-62.828944347,7.505027085],[0.675020638,-0.047590368,0.079986947,0.731904627],[0,0,0,1],[9E+09,9E+09,9E+09,9E+09,9E+09,9E+09]];
    CONST robtarget Con_340:=[[175.230586514,-33.267770234,0.694727348],[0.66884149,-0.077783626,0.109808671,0.731124356],[0,0,0,1],[9E+09,9E+09,9E+09,9E+09,9E+09,9E+09]];
    CONST robtarget Con_350:=[[173.914122015,-20.027548797,-3.086383197],[0.666275035,-0.086634844,0.118897307,0.731050895],[0,0,0,1],[9E+09,9E+09,9E+09,9E+09,9E+09,9E+09]];
    CONST robtarget Con_360:=[[172.187743436,-3.581680271,-8.24430743],[0.663178379,-0.095334203,0.128138196,0.731222559],[0,0,0,1],[9E+09,9E+09,9E+09,9E+09,9E+09,9E+09]];
    CONST robtarget Con_370:=[[171.065027221,6.614957341,-11.657747544],[0.661286765,-0.099740344,0.133005032,0.731478872],[0,0,0,1],[9E+09,9E+09,9E+09,9E+09,9E+09,9E+09]];
    CONST robtarget Con_380:=[[169.705716929,18.480973126,-15.809132933],[0.659080069,-0.104153349,0.13806505,0.731917745],[0,0,0,1],[9E+09,9E+09,9E+09,9E+09,9E+09,9E+09]];
    CONST robtarget Con_390:=[[168.316647478,30.103101955,-20.040376869],[0.656891012,-0.107854262,0.142514724,0.73249656],[0,0,0,1],[9E+09,9E+09,9E+09,9E+09,9E+09,9E+09]];
    CONST robtarget Con_400:=[[166.543823848,44.249477068,-25.386000274],[0.654165899,-0.111650869,0.147380232,0.733403113],[0,0,0,1],[9E+09,9E+09,9E+09,9E+09,9E+09,9E+09]];
    CONST robtarget Con_410:=[[164.876552143,56.900000803,-30.327636979],[0.651610512,-0.114536414,0.151377118,0.734418218],[0,0,0,1],[9E+09,9E+09,9E+09,9E+09,9E+09,9E+09]];
    CONST robtarget Con_420:=[[163.037520807,70.162534848,-35.655969883],[0.648777542,-0.117101246,0.155280974,0.73570566],[0,0,0,1],[9E+09,9E+09,9E+09,9E+09,9E+09,9E+09]];
    CONST robtarget Con_30:=[[200.00005472,-551.158225865,-88.527467846],[0.634133695,0.312848991,-0.312560668,0.634275804],[0,-1,1,0],[9E+09,9E+09,9E+09,9E+09,9E+09,9E+09]];
    CONST robtarget Con_440:=[[157.096307132,106.775473629,-46.27509895],[0.58303405,-0.109888923,0.191745437,0.781811619],[0,0,0,1],[9E+09,9E+09,9E+09,9E+09,9E+09,9E+09]];
    CONST robtarget Con_450:=[[150.648978166,119.286589367,-52.471354293],[0.47074561,-0.098382093,0.237866386,0.843883355],[0,0,1,1],[9E+09,9E+09,9E+09,9E+09,9E+09,9E+09]];
    CONST robtarget Con_460:=[[143.724533585,127.096786841,-56.624499986],[0.386615909,-0.082035042,0.259666215,0.881119656],[0,0,1,1],[9E+09,9E+09,9E+09,9E+09,9E+09,9E+09]];
    CONST robtarget Con_470:=[[130.330544937,137.18843292,-62.128190813],[0.31779168,-0.06858341,0.273418247,0.905288477],[0,0,1,1],[9E+09,9E+09,9E+09,9E+09,9E+09,9E+09]];
    CONST robtarget Con_480:=[[118.483347543,144.537440829,-66.250564627],[0.276838465,-0.061788855,0.280368946,0.917025548],[0,0,1,1],[9E+09,9E+09,9E+09,9E+09,9E+09,9E+09]];
    CONST robtarget Con_490:=[[106.060784114,150.916477899,-69.906430657],[0.238586474,-0.05468288,0.285668113,0.926541962],[0,0,1,1],[9E+09,9E+09,9E+09,9E+09,9E+09,9E+09]];
    CONST robtarget Con_500:=[[94.010851589,156.064307862,-72.904751563],[0.205101845,-0.047971076,0.289479141,0.933720427],[0,0,1,1],[9E+09,9E+09,9E+09,9E+09,9E+09,9E+09]];
    CONST robtarget Con_510:=[[81.965076033,160.356717918,-75.43566318],[0.174479478,-0.04147194,0.292352052,0.939344062],[0,0,1,1],[9E+09,9E+09,9E+09,9E+09,9E+09,9E+09]];
    CONST robtarget Last_20:=[[195.048135633,-586.860489021,-123.704781043],[-0.000000016,0.000000073,-0.46295826,0.886380082],[0,-2,3,0],[9E+09,9E+09,9E+09,9E+09,9E+09,9E+09]];
    CONST robtarget Con_530:=[[51.193155532,168.15560706,-80.102691439],[0.104925833,-0.025667913,0.296935974,0.94876802],[0,0,1,1],[9E+09,9E+09,9E+09,9E+09,9E+09,9E+09]];
    CONST robtarget Con_540:=[[40.744816596,169.911065218,-81.164072048],[0.083177113,-0.020403077,0.297859151,0.950760332],[0,0,1,1],[9E+09,9E+09,9E+09,9E+09,9E+09,9E+09]];
    CONST robtarget Con_550:=[[19.400325474,170.867618687,-80.674001449],[0,0.000000035,0.369539494,0.929215025],[0,0,1,1],[9E+09,9E+09,9E+09,9E+09,9E+09,9E+09]];
    CONST robtarget Con_560:=[[2.586940581,170.867619128,-80.674000339],[0,0.000000035,0.369539494,0.929215025],[0,0,1,1],[9E+09,9E+09,9E+09,9E+09,9E+09,9E+09]];
    CONST robtarget Con_570:=[[-27.099155839,170.867619907,-80.673998381],[0,0.000000035,0.369539494,0.929215025],[0,0,1,1],[9E+09,9E+09,9E+09,9E+09,9E+09,9E+09]];
    CONST robtarget Con_580:=[[-64.315106976,165.33597811,-78.405387263],[0.133349913,-0.032289351,-0.295370437,-0.94547951],[-1,-1,2,1],[9E+09,9E+09,9E+09,9E+09,9E+09,9E+09]];
    CONST robtarget Con_590:=[[-107.55620446,150.210439939,-69.498455667],[0.242978993,-0.055531199,-0.285113145,-0.925520389],[-1,-1,2,1],[9E+09,9E+09,9E+09,9E+09,9E+09,9E+09]];
    CONST robtarget Con_600:=[[-127.235661403,139.245885525,-63.272037935],[0.306607867,-0.066823906,-0.27545973,-0.908651814],[-1,-1,2,1],[9E+09,9E+09,9E+09,9E+09,9E+09,9E+09]];
    CONST robtarget Last_10:=[[-142.521139439,-586.860484387,-123.704730918],[0.000000016,0.000000073,-0.46295826,0.886380082],[-1,0,1,0],[9E+09,9E+09,9E+09,9E+09,9E+09,9E+09]];
    CONST robtarget Con_20:=[[200.000053486,-562.541878275,-102.708516773],[0.641627386,0.297177273,-0.297177238,0.641627349],[0,-1,1,0],[9E+09,9E+09,9E+09,9E+09,9E+09,9E+09]];
    CONST robtarget Con_630:=[[-158.266587633,102.773171095,-44.601832483],[0.616052419,-0.090410149,-0.159155117,-0.766142984],[-1,-1,2,1],[9E+09,9E+09,9E+09,9E+09,9E+09,9E+09]];
    CONST robtarget Con_640:=[[-162.003694891,77.316481098,-38.587354653],[0.647185108,-0.118284489,-0.15726657,-0.736496735],[-1,-1,3,1],[9E+09,9E+09,9E+09,9E+09,9E+09,9E+09]];
    CONST robtarget Con_650:=[[-166.462564633,44.879254465,-25.628518843],[0.654042118,-0.111804527,-0.147585515,-0.73344882],[-1,-1,3,1],[9E+09,9E+09,9E+09,9E+09,9E+09,9E+09]];
    CONST robtarget Con_660:=[[-169.83567573,17.366882463,-15.411774128],[0.65928718,-0.103771759,-0.13761729,-0.731869741],[-1,-1,3,1],[9E+09,9E+09,9E+09,9E+09,9E+09,9E+09]];
    CONST robtarget Con_670:=[[-173.446009451,-15.472041963,-4.467813294],[0.66540886,-0.089270527,-0.121656819,-0.731068697],[-1,-1,3,1],[9E+09,9E+09,9E+09,9E+09,9E+09,9E+09]];
    CONST robtarget Con_680:=[[-176.624550081,-48.056835414,4.430975485],[0.671843909,-0.065013038,-0.09703582,-0.7314254],[-1,-1,3,1],[9E+09,9E+09,9E+09,9E+09,9E+09,9E+09]];
    CONST robtarget Con_690:=[[-179.170760408,-77.765992815,9.702045768],[0.6783366,-0.022014249,-0.05536715,-0.73233142],[-1,-1,3,1],[9E+09,9E+09,9E+09,9E+09,9E+09,9E+09]];
    CONST robtarget Con_700:=[[-181.305159966,-102.322040378,13.816606291],[0.669561043,-0.074501736,-0.106600762,-0.731282284],[-1,-1,3,1],[9E+09,9E+09,9E+09,9E+09,9E+09,9E+09]];
    CONST robtarget Con_710:=[[-184.328477669,-133.584297025,22.698059205],[0.667319114,-0.090534635,-0.12105633,-0.729269529],[-1,-1,3,1],[9E+09,9E+09,9E+09,9E+09,9E+09,9E+09]];
    CONST robtarget Con_720:=[[-188.351452181,-174.042967383,36.742971591],[0.662764432,-0.11710002,-0.14510734,-0.725241169],[-1,-1,3,1],[9E+09,9E+09,9E+09,9E+09,9E+09,9E+09]];
    CONST robtarget Con_730:=[[-192.1683216,-210.752572402,52.952743751],[0.655614461,-0.150068462,-0.17509046,-0.719021881],[-1,-1,3,1],[9E+09,9E+09,9E+09,9E+09,9E+09,9E+09]];
    CONST robtarget Con_740:=[[-195.272963674,-238.843377223,68.681316885],[0.646166031,-0.18465933,-0.20670734,-0.711085415],[-1,-1,3,1],[9E+09,9E+09,9E+09,9E+09,9E+09,9E+09]];
    CONST robtarget Con_750:=[[-198.035689462,-261.832436248,84.700811019],[0.635328635,-0.214892904,-0.234824147,-0.70358808],[-1,-1,3,1],[9E+09,9E+09,9E+09,9E+09,9E+09,9E+09]];
    CONST robtarget Con_760:=[[-199.999925879,-290.464167255,101.923821981],[0.680314092,-0.192802342,-0.192802292,-0.680314097],[-1,-1,3,1],[9E+09,9E+09,9E+09,9E+09,9E+09,9E+09]];
    CONST robtarget Con_770:=[[-199.9999255,-323.252878302,120.702108677],[0.693574212,-0.137676477,-0.137676427,-0.693574222],[-1,-1,3,1],[9E+09,9E+09,9E+09,9E+09,9E+09,9E+09]];
    CONST robtarget Con_780:=[[-199.999925781,-359.604985793,130.892623305],[0.705647237,-0.045408906,-0.045408858,-0.705647252],[-1,-1,3,1],[9E+09,9E+09,9E+09,9E+09,9E+09,9E+09]];
    CONST robtarget Con_790:=[[-199.999926819,-393.912161454,128.803944419],[0.700292992,0.097927033,0.097927077,-0.700293017],[-1,-1,3,1],[9E+09,9E+09,9E+09,9E+09,9E+09,9E+09]];
    CONST robtarget Con_820:=[[-199.999933423,-460.601994969,55.218950295],[0.611283812,0.355432225,0.355432256,-0.611283851],[-1,0,2,0],[9E+09,9E+09,9E+09,9E+09,9E+09,9E+09]];
    CONST robtarget Con_830:=[[-199.999940642,-512.732986741,-33.487590507],[0.626765351,0.327360902,0.327360934,-0.626765389],[-1,0,2,0],[9E+09,9E+09,9E+09,9E+09,9E+09,9E+09]];
    CONST robtarget Con_840:=[[-199.999945851,-556.318627929,-95.127641129],[0.637110507,0.306741207,0.306741241,-0.637110544],[-1,0,2,0],[9E+09,9E+09,9E+09,9E+09,9E+09,9E+09]];
    CONST robtarget Con_850:=[[-199.999947551,-573.095410485,-114.220901185],[0.654581876,0.267436974,0.26743701,-0.654581911],[-1,0,2,0],[9E+09,9E+09,9E+09,9E+09,9E+09,9E+09]];
    CONST robtarget Con_860:=[[-199.999948196,-580.967121247,-120.87051345],[0.677204022,0.203456834,0.203456873,-0.677204053],[-1,0,2,0],[9E+09,9E+09,9E+09,9E+09,9E+09,9E+09]];
    CONST robtarget Con_610:=[[-143.002888572,127.755720301,-56.981193482],[0.379115268,-0.080518646,-0.26131325,-0.884027006],[-1,-1,2,1],[9E+09,9E+09,9E+09,9E+09,9E+09,9E+09]];
    CONST robtarget Con_620:=[[-153.368513821,115.05495469,-50.293347526],[0.511910998,-0.105361505,-0.224363229,-0.822500593],[-1,-1,2,1],[9E+09,9E+09,9E+09,9E+09,9E+09,9E+09]];
    CONST robtarget Con_430:=[[160.452539045,88.477140471,-41.732741555],[0.655810432,-0.058206333,0.106035754,0.745171872],[0,0,0,1],[9E+09,9E+09,9E+09,9E+09,9E+09,9E+09]];
    CONST robtarget Con_800:=[[-199.999928557,-421.768055651,113.532077086],[0.662167022,0.248062096,0.248061639,-0.662167241],[-1,0,2,0],[9E+09,9E+09,9E+09,9E+09,9E+09,9E+09]];
    CONST robtarget Con_330:=[[176.76658024,-49.611972612,4.78874382],[0.672170284,-0.063433206,0.095475683,0.73146957],[0,0,0,1],[9E+09,9E+09,9E+09,9E+09,9E+09,9E+09]];
    CONST robtarget Con_40:=[[200.000055921,-541.142954729,-74.297775882],[0.626765389,0.327360934,-0.327360902,0.626765351],[0,-1,1,0],[9E+09,9E+09,9E+09,9E+09,9E+09,9E+09]];
    CONST robtarget Con_150:=[[200.000073085,-395.995547818,128.17542892],[0.698730559,0.10851557,-0.108515526,0.698730533],[0,-1,1,0],[9E+09,9E+09,9E+09,9E+09,9E+09,9E+09]];
    CONST robtarget Con_60:=[[200.000058864,-516.819515009,-39.357792523],[0.626765389,0.327360934,-0.327360902,0.626765351],[0,-1,1,0],[9E+09,9E+09,9E+09,9E+09,9E+09,9E+09]];
    CONST robtarget Con_70:=[[200.000060942,-500.675934872,-14.27735974],[0.615030116,0.348909718,-0.348909687,0.615030077],[0,-1,1,0],[9E+09,9E+09,9E+09,9E+09,9E+09,9E+09]];
    CONST robtarget Con_80:=[[200.000062389,-490.223041219,3.50034115],[0.612861942,0.352704232,-0.352704201,0.612861902],[0,-1,1,0],[9E+09,9E+09,9E+09,9E+09,9E+09,9E+09]];
    CONST robtarget Con_90:=[[200.000064208,-477.296059885,25.939514748],[0.611714679,0.354690269,-0.354690238,0.611714639],[0,-1,1,0],[9E+09,9E+09,9E+09,9E+09,9E+09,9E+09]];
    CONST robtarget Con_50:=[[200.000057578,-527.44428565,-54.61999695],[0.626765389,0.327360934,-0.327360902,0.626765351],[0,-1,1,0],[9E+09,9E+09,9E+09,9E+09,9E+09,9E+09]];
    CONST robtarget Con_10:=[[200.000052357,-574.121968432,-115.213504775],[0.656521822,0.262638781,-0.262638745,0.656521787],[0,-1,1,0],[9E+09,9E+09,9E+09,9E+09,9E+09,9E+09]];
!***********************************************************
    !
    ! Módulo:  Module1
    !
    ! Descripción:
    !   <Introduzca la descripción aquí>
    !
    ! Autor: David
    !
    ! Versión: 1.0
    !
    !***********************************************************


    !***********************************************************
    !
    ! Procedimiento Main
    !
    !   Este es el punto de entrada de su programa
    !
    !***********************************************************
    PROC main()
        CUTTING_ROUTINE:
        WaitDI Holes_Cut,1;
        Hole1;
        Hole2;
        Hole3;
        PulseDO Holes_Done;
        WaitDI Contour_Cut,1;
        Contour;
        PulseDO Contour_Done;
        GOTO CUTTING_ROUTINE;
    ENDPROC
    PROC Hole1()
        MoveJ Target_30,v300,fine,Ultrasonic_Cutter_TCP\WObj:=Workobject_2;
        MoveJ Target_40,v300,fine,Ultrasonic_Cutter_TCP\WObj:=Workobject_2;
        MoveJ H1_10,v300,fine,Ultrasonic_Cutter_TCP\WObj:=Workobject_2;
        MoveJ H1_20,v300,fine,Ultrasonic_Cutter_TCP\WObj:=Workobject_2;
        MoveJ H1_30,v300,fine,Ultrasonic_Cutter_TCP\WObj:=Workobject_2;
        MoveJ H1_40,v300,fine,Ultrasonic_Cutter_TCP\WObj:=Workobject_2;
        MoveJ H1_50,v300,fine,Ultrasonic_Cutter_TCP\WObj:=Workobject_2;
        MoveJ H1_60,v300,fine,Ultrasonic_Cutter_TCP\WObj:=Workobject_2;
        MoveJ H1_70,v300,fine,Ultrasonic_Cutter_TCP\WObj:=Workobject_2;
        MoveJ H1_80,v300,fine,Ultrasonic_Cutter_TCP\WObj:=Workobject_2;
        MoveJ H1_90,v300,fine,Ultrasonic_Cutter_TCP\WObj:=Workobject_2;
        MoveJ H1_100,v300,fine,Ultrasonic_Cutter_TCP\WObj:=Workobject_2;
        MoveJ H1_110,v300,fine,Ultrasonic_Cutter_TCP\WObj:=Workobject_2;
        MoveJ H1_120,v300,fine,Ultrasonic_Cutter_TCP\WObj:=Workobject_2;
        MoveJ H1_130,v300,fine,Ultrasonic_Cutter_TCP\WObj:=Workobject_2;
        MoveJ H1_140,v300,fine,Ultrasonic_Cutter_TCP\WObj:=Workobject_2;
        MoveJ H1_150,v300,fine,Ultrasonic_Cutter_TCP\WObj:=Workobject_2;
        MoveJ H1_160,v300,fine,Ultrasonic_Cutter_TCP\WObj:=Workobject_2;
        MoveJ H1_170,v300,fine,Ultrasonic_Cutter_TCP\WObj:=Workobject_2;
        MoveJ H1_180,v300,fine,Ultrasonic_Cutter_TCP\WObj:=Workobject_2;
        MoveJ H1_190,v300,fine,Ultrasonic_Cutter_TCP\WObj:=Workobject_2;
        MoveJ H1_200,v300,fine,Ultrasonic_Cutter_TCP\WObj:=Workobject_2;
        MoveJ H1_210,v300,fine,Ultrasonic_Cutter_TCP\WObj:=Workobject_2;
        MoveJ H1_220,v300,fine,Ultrasonic_Cutter_TCP\WObj:=Workobject_2;
        MoveJ H1_230,v300,fine,Ultrasonic_Cutter_TCP\WObj:=Workobject_2;
        MoveJ H1_240,v300,fine,Ultrasonic_Cutter_TCP\WObj:=Workobject_2;
        MoveJ H1_250,v300,fine,Ultrasonic_Cutter_TCP\WObj:=Workobject_2;
        MoveJ H1_260,v300,fine,Ultrasonic_Cutter_TCP\WObj:=Workobject_2;
        MoveJ H1_270,v300,fine,Ultrasonic_Cutter_TCP\WObj:=Workobject_2;
        MoveJ H1_280,v300,fine,Ultrasonic_Cutter_TCP\WObj:=Workobject_2;
        MoveJ H1_290,v300,fine,Ultrasonic_Cutter_TCP\WObj:=Workobject_2;
        MoveJ H1_300,v300,fine,Ultrasonic_Cutter_TCP\WObj:=Workobject_2;
        MoveJ H1_310,v300,fine,Ultrasonic_Cutter_TCP\WObj:=Workobject_2;
        MoveJ H1_320,v300,fine,Ultrasonic_Cutter_TCP\WObj:=Workobject_2;
        MoveJ H1_330,v300,fine,Ultrasonic_Cutter_TCP\WObj:=Workobject_2;
        MoveJ H1_340,v300,fine,Ultrasonic_Cutter_TCP\WObj:=Workobject_2;
        MoveJ H1_350,v300,fine,Ultrasonic_Cutter_TCP\WObj:=Workobject_2;
        MoveJ H1_360,v300,fine,Ultrasonic_Cutter_TCP\WObj:=Workobject_2;
        MoveJ H1_370,v300,fine,Ultrasonic_Cutter_TCP\WObj:=Workobject_2;
        MoveJ H1_380,v300,fine,Ultrasonic_Cutter_TCP\WObj:=Workobject_2;
        MoveJ H1_390,v300,fine,Ultrasonic_Cutter_TCP\WObj:=Workobject_2;
        MoveJ H1_400,v300,fine,Ultrasonic_Cutter_TCP\WObj:=Workobject_2;
        MoveJ H1_410,v300,fine,Ultrasonic_Cutter_TCP\WObj:=Workobject_2;
        MoveJ H1_420,v300,fine,Ultrasonic_Cutter_TCP\WObj:=Workobject_2;
        MoveJ H1_430,v300,fine,Ultrasonic_Cutter_TCP\WObj:=Workobject_2;
        MoveJ H1_440,v300,fine,Ultrasonic_Cutter_TCP\WObj:=Workobject_2;
        MoveJ H1_450,v300,fine,Ultrasonic_Cutter_TCP\WObj:=Workobject_2;
        MoveJ H1_460,v300,fine,Ultrasonic_Cutter_TCP\WObj:=Workobject_2;
        MoveJ H1_470,v300,fine,Ultrasonic_Cutter_TCP\WObj:=Workobject_2;
        MoveJ H1_480,v300,fine,Ultrasonic_Cutter_TCP\WObj:=Workobject_2;
        MoveJ H1_490,v300,fine,Ultrasonic_Cutter_TCP\WObj:=Workobject_2;
        MoveJ H1_500,v300,fine,Ultrasonic_Cutter_TCP\WObj:=Workobject_2;
        MoveJ H1_510,v300,fine,Ultrasonic_Cutter_TCP\WObj:=Workobject_2;
        MoveJ H1_520,v300,fine,Ultrasonic_Cutter_TCP\WObj:=Workobject_2;
        MoveJ Target_40,v300,fine,Ultrasonic_Cutter_TCP\WObj:=Workobject_2;
        MoveJ Target_30,v300,fine,Ultrasonic_Cutter_TCP\WObj:=Workobject_2;
    ENDPROC
    PROC Hole2()
        MoveJ Target_30,v300,fine,Ultrasonic_Cutter_TCP\WObj:=Workobject_2;
        MoveJ Target_50,v300,fine,Ultrasonic_Cutter_TCP\WObj:=Workobject_2;
        MoveJ H2_10,v300,fine,Ultrasonic_Cutter_TCP\WObj:=Workobject_2;
        MoveJ H2_20,v300,fine,Ultrasonic_Cutter_TCP\WObj:=Workobject_2;
        MoveJ H2_30,v300,fine,Ultrasonic_Cutter_TCP\WObj:=Workobject_2;
        MoveJ H2_40,v300,fine,Ultrasonic_Cutter_TCP\WObj:=Workobject_2;
        MoveJ H2_50,v300,fine,Ultrasonic_Cutter_TCP\WObj:=Workobject_2;
        MoveJ H2_60,v300,fine,Ultrasonic_Cutter_TCP\WObj:=Workobject_2;
        MoveJ H2_70,v300,fine,Ultrasonic_Cutter_TCP\WObj:=Workobject_2;
        MoveJ H2_80,v300,fine,Ultrasonic_Cutter_TCP\WObj:=Workobject_2;
        MoveJ H2_90,v300,fine,Ultrasonic_Cutter_TCP\WObj:=Workobject_2;
        MoveJ H2_100,v300,fine,Ultrasonic_Cutter_TCP\WObj:=Workobject_2;
        MoveJ H2_110,v300,fine,Ultrasonic_Cutter_TCP\WObj:=Workobject_2;
        MoveJ H2_120,v300,fine,Ultrasonic_Cutter_TCP\WObj:=Workobject_2;
        MoveJ H2_130,v300,fine,Ultrasonic_Cutter_TCP\WObj:=Workobject_2;
        MoveJ H2_140,v300,fine,Ultrasonic_Cutter_TCP\WObj:=Workobject_2;
        MoveJ H2_150,v300,fine,Ultrasonic_Cutter_TCP\WObj:=Workobject_2;
        MoveJ H2_160,v300,fine,Ultrasonic_Cutter_TCP\WObj:=Workobject_2;
        MoveJ H2_170,v300,fine,Ultrasonic_Cutter_TCP\WObj:=Workobject_2;
        MoveJ H2_180,v300,fine,Ultrasonic_Cutter_TCP\WObj:=Workobject_2;
        MoveJ H2_190,v300,fine,Ultrasonic_Cutter_TCP\WObj:=Workobject_2;
        MoveJ H2_200,v300,fine,Ultrasonic_Cutter_TCP\WObj:=Workobject_2;
        MoveJ H2_210,v300,fine,Ultrasonic_Cutter_TCP\WObj:=Workobject_2;
        MoveJ H2_220,v300,fine,Ultrasonic_Cutter_TCP\WObj:=Workobject_2;
        MoveJ H2_230,v300,fine,Ultrasonic_Cutter_TCP\WObj:=Workobject_2;
        MoveJ Target_50,v300,fine,Ultrasonic_Cutter_TCP\WObj:=Workobject_2;
        MoveJ Target_30,v300,fine,Ultrasonic_Cutter_TCP\WObj:=Workobject_2;
    ENDPROC
    PROC Hole3()
        MoveJ Target_30,v300,fine,Ultrasonic_Cutter_TCP\WObj:=Workobject_2;
        MoveJ Target_60,v300,fine,Ultrasonic_Cutter_TCP\WObj:=Workobject_2;
        MoveJ H3_10,v300,fine,Ultrasonic_Cutter_TCP\WObj:=Workobject_2;
        MoveJ H3_20,v300,fine,Ultrasonic_Cutter_TCP\WObj:=Workobject_2;
        MoveJ H3_30,v300,fine,Ultrasonic_Cutter_TCP\WObj:=Workobject_2;
        MoveJ H3_40,v300,fine,Ultrasonic_Cutter_TCP\WObj:=Workobject_2;
        MoveJ H3_50,v300,fine,Ultrasonic_Cutter_TCP\WObj:=Workobject_2;
        MoveJ H3_60,v300,fine,Ultrasonic_Cutter_TCP\WObj:=Workobject_2;
        MoveJ H3_70,v300,fine,Ultrasonic_Cutter_TCP\WObj:=Workobject_2;
        MoveJ H3_80,v300,fine,Ultrasonic_Cutter_TCP\WObj:=Workobject_2;
        MoveJ H3_90,v300,fine,Ultrasonic_Cutter_TCP\WObj:=Workobject_2;
        MoveJ H3_100,v300,fine,Ultrasonic_Cutter_TCP\WObj:=Workobject_2;
        MoveJ H3_110,v300,fine,Ultrasonic_Cutter_TCP\WObj:=Workobject_2;
        MoveJ H3_120,v300,fine,Ultrasonic_Cutter_TCP\WObj:=Workobject_2;
        MoveJ H3_130,v300,fine,Ultrasonic_Cutter_TCP\WObj:=Workobject_2;
        MoveJ H3_140,v300,fine,Ultrasonic_Cutter_TCP\WObj:=Workobject_2;
        MoveJ H3_150,v300,fine,Ultrasonic_Cutter_TCP\WObj:=Workobject_2;
        MoveJ H3_160,v300,fine,Ultrasonic_Cutter_TCP\WObj:=Workobject_2;
        MoveJ H3_170,v300,fine,Ultrasonic_Cutter_TCP\WObj:=Workobject_2;
        MoveJ H3_180,v300,fine,Ultrasonic_Cutter_TCP\WObj:=Workobject_2;
        MoveJ H3_190,v300,fine,Ultrasonic_Cutter_TCP\WObj:=Workobject_2;
        MoveJ H3_200,v300,fine,Ultrasonic_Cutter_TCP\WObj:=Workobject_2;
        MoveJ H3_210,v300,fine,Ultrasonic_Cutter_TCP\WObj:=Workobject_2;
        MoveJ H3_220,v300,fine,Ultrasonic_Cutter_TCP\WObj:=Workobject_2;
        MoveJ H3_230,v300,fine,Ultrasonic_Cutter_TCP\WObj:=Workobject_2;
        MoveJ H3_240,v300,fine,Ultrasonic_Cutter_TCP\WObj:=Workobject_2;
        MoveJ H3_250,v300,fine,Ultrasonic_Cutter_TCP\WObj:=Workobject_2;
        MoveJ H3_260,v300,fine,Ultrasonic_Cutter_TCP\WObj:=Workobject_2;
        MoveJ Target_60,v300,fine,Ultrasonic_Cutter_TCP\WObj:=Workobject_2;
        MoveJ Target_30,v300,fine,Ultrasonic_Cutter_TCP\WObj:=Workobject_2;
    ENDPROC
    PROC Contour()
        MoveJ Target_30,v300,fine,Ultrasonic_Cutter_TCP\WObj:=Workobject_2;
        MoveJ Target_70,v300,fine,Ultrasonic_Cutter_TCP\WObj:=Workobject_2;
        MoveJ Con_10,v300,fine,Ultrasonic_Cutter_TCP\WObj:=Workobject_2;
        MoveJ Con_20,v300,fine,Ultrasonic_Cutter_TCP\WObj:=Workobject_2;
        MoveJ Con_30,v300,fine,Ultrasonic_Cutter_TCP\WObj:=Workobject_2;
        MoveJ Con_40,v300,fine,Ultrasonic_Cutter_TCP\WObj:=Workobject_2;
        MoveJ Con_50,v300,fine,Ultrasonic_Cutter_TCP\WObj:=Workobject_2;
        MoveJ Con_60,v300,fine,Ultrasonic_Cutter_TCP\WObj:=Workobject_2;
        MoveJ Con_70,v300,fine,Ultrasonic_Cutter_TCP\WObj:=Workobject_2;
        MoveJ Con_80,v300,fine,Ultrasonic_Cutter_TCP\WObj:=Workobject_2;
        MoveJ Con_90,v300,fine,Ultrasonic_Cutter_TCP\WObj:=Workobject_2;
        MoveJ Con_100,v300,fine,Ultrasonic_Cutter_TCP\WObj:=Workobject_2;
        MoveJ Con_110,v300,fine,Ultrasonic_Cutter_TCP\WObj:=Workobject_2;
        MoveJ Con_130,v300,fine,Ultrasonic_Cutter_TCP\WObj:=Workobject_2;
        MoveJ Con_140,v300,fine,Ultrasonic_Cutter_TCP\WObj:=Workobject_2;
        MoveJ Con_150,v300,fine,Ultrasonic_Cutter_TCP\WObj:=Workobject_2;
        MoveJ Con_160,v300,fine,Ultrasonic_Cutter_TCP\WObj:=Workobject_2;
        MoveJ Con_170,v300,fine,Ultrasonic_Cutter_TCP\WObj:=Workobject_2;
        MoveJ Con_180,v300,fine,Ultrasonic_Cutter_TCP\WObj:=Workobject_2;
        MoveJ Con_190,v300,fine,Ultrasonic_Cutter_TCP\WObj:=Workobject_2;
        MoveJ Con_200,v300,fine,Ultrasonic_Cutter_TCP\WObj:=Workobject_2;
        MoveJ Con_210,v300,fine,Ultrasonic_Cutter_TCP\WObj:=Workobject_2;
        MoveJ Con_220,v300,fine,Ultrasonic_Cutter_TCP\WObj:=Workobject_2;
        MoveJ Con_230,v300,fine,Ultrasonic_Cutter_TCP\WObj:=Workobject_2;
        MoveJ Con_240,v300,fine,Ultrasonic_Cutter_TCP\WObj:=Workobject_2;
        MoveJ Con_250,v300,fine,Ultrasonic_Cutter_TCP\WObj:=Workobject_2;
        MoveJ Con_260,v300,fine,Ultrasonic_Cutter_TCP\WObj:=Workobject_2;
        MoveJ Con_270,v300,fine,Ultrasonic_Cutter_TCP\WObj:=Workobject_2;
        MoveJ Con_280,v300,fine,Ultrasonic_Cutter_TCP\WObj:=Workobject_2;
        MoveJ Con_290,v300,fine,Ultrasonic_Cutter_TCP\WObj:=Workobject_2;
        MoveJ Con_300,v300,fine,Ultrasonic_Cutter_TCP\WObj:=Workobject_2;
        MoveJ Con_310,v300,fine,Ultrasonic_Cutter_TCP\WObj:=Workobject_2;
        MoveJ Con_320,v300,fine,Ultrasonic_Cutter_TCP\WObj:=Workobject_2;
        MoveJ Con_330,v300,fine,Ultrasonic_Cutter_TCP\WObj:=Workobject_2;
        MoveJ Con_340,v300,fine,Ultrasonic_Cutter_TCP\WObj:=Workobject_2;
        MoveJ Con_350,v300,fine,Ultrasonic_Cutter_TCP\WObj:=Workobject_2;
        MoveJ Con_360,v300,fine,Ultrasonic_Cutter_TCP\WObj:=Workobject_2;
        MoveJ Con_370,v300,fine,Ultrasonic_Cutter_TCP\WObj:=Workobject_2;
        MoveJ Con_380,v300,fine,Ultrasonic_Cutter_TCP\WObj:=Workobject_2;
        MoveJ Con_390,v300,fine,Ultrasonic_Cutter_TCP\WObj:=Workobject_2;
        MoveJ Con_400,v300,fine,Ultrasonic_Cutter_TCP\WObj:=Workobject_2;
        MoveJ Con_410,v300,fine,Ultrasonic_Cutter_TCP\WObj:=Workobject_2;
        MoveJ Con_420,v300,fine,Ultrasonic_Cutter_TCP\WObj:=Workobject_2;
        MoveJ Con_430,v300,fine,Ultrasonic_Cutter_TCP\WObj:=Workobject_2;
        MoveJ Con_440,v300,fine,Ultrasonic_Cutter_TCP\WObj:=Workobject_2;
        MoveJ Con_450,v300,fine,Ultrasonic_Cutter_TCP\WObj:=Workobject_2;
        MoveJ Con_460,v300,fine,Ultrasonic_Cutter_TCP\WObj:=Workobject_2;
        MoveJ Con_470,v300,fine,Ultrasonic_Cutter_TCP\WObj:=Workobject_2;
        MoveJ Con_480,v300,fine,Ultrasonic_Cutter_TCP\WObj:=Workobject_2;
        MoveJ Con_490,v300,fine,Ultrasonic_Cutter_TCP\WObj:=Workobject_2;
        MoveJ Con_500,v300,fine,Ultrasonic_Cutter_TCP\WObj:=Workobject_2;
        MoveJ Con_510,v300,fine,Ultrasonic_Cutter_TCP\WObj:=Workobject_2;
        MoveJ Con_520,v300,fine,Ultrasonic_Cutter_TCP\WObj:=Workobject_2;
        MoveJ Con_530,v300,fine,Ultrasonic_Cutter_TCP\WObj:=Workobject_2;
        MoveJ Con_540,v300,fine,Ultrasonic_Cutter_TCP\WObj:=Workobject_2;
        MoveJ Con_550,v300,fine,Ultrasonic_Cutter_TCP\WObj:=Workobject_2;
        MoveJ Con_560,v300,fine,Ultrasonic_Cutter_TCP\WObj:=Workobject_2;
        MoveJ Con_570,v300,fine,Ultrasonic_Cutter_TCP\WObj:=Workobject_2;
        MoveJ Con_580,v300,fine,Ultrasonic_Cutter_TCP\WObj:=Workobject_2;
        MoveJ Con_590,v300,fine,Ultrasonic_Cutter_TCP\WObj:=Workobject_2;
        MoveJ Con_600,v300,fine,Ultrasonic_Cutter_TCP\WObj:=Workobject_2;
        MoveJ Con_610,v300,fine,Ultrasonic_Cutter_TCP\WObj:=Workobject_2;
        MoveJ Con_620,v300,fine,Ultrasonic_Cutter_TCP\WObj:=Workobject_2;
        MoveJ Con_630,v300,fine,Ultrasonic_Cutter_TCP\WObj:=Workobject_2;
        MoveJ Con_640,v300,fine,Ultrasonic_Cutter_TCP\WObj:=Workobject_2;
        MoveJ Con_650,v300,fine,Ultrasonic_Cutter_TCP\WObj:=Workobject_2;
        MoveJ Con_660,v300,fine,Ultrasonic_Cutter_TCP\WObj:=Workobject_2;
        MoveJ Con_670,v300,fine,Ultrasonic_Cutter_TCP\WObj:=Workobject_2;
        MoveJ Con_680,v300,fine,Ultrasonic_Cutter_TCP\WObj:=Workobject_2;
        MoveJ Con_690,v300,fine,Ultrasonic_Cutter_TCP\WObj:=Workobject_2;
        MoveJ Con_700,v300,fine,Ultrasonic_Cutter_TCP\WObj:=Workobject_2;
        MoveJ Con_710,v300,fine,Ultrasonic_Cutter_TCP\WObj:=Workobject_2;
        MoveJ Con_720,v300,fine,Ultrasonic_Cutter_TCP\WObj:=Workobject_2;
        MoveJ Con_730,v300,fine,Ultrasonic_Cutter_TCP\WObj:=Workobject_2;
        MoveJ Con_740,v300,fine,Ultrasonic_Cutter_TCP\WObj:=Workobject_2;
        MoveJ Con_750,v300,fine,Ultrasonic_Cutter_TCP\WObj:=Workobject_2;
        MoveJ Con_760,v300,fine,Ultrasonic_Cutter_TCP\WObj:=Workobject_2;
        MoveJ Con_770,v300,fine,Ultrasonic_Cutter_TCP\WObj:=Workobject_2;
        MoveJ Con_780,v300,fine,Ultrasonic_Cutter_TCP\WObj:=Workobject_2;
        MoveJ Con_790,v300,fine,Ultrasonic_Cutter_TCP\WObj:=Workobject_2;
        MoveJ Con_800,v300,fine,Ultrasonic_Cutter_TCP\WObj:=Workobject_2;
        MoveJ Con_820,v300,fine,Ultrasonic_Cutter_TCP\WObj:=Workobject_2;
        MoveJ Con_830,v300,fine,Ultrasonic_Cutter_TCP\WObj:=Workobject_2;
        MoveJ Con_840,v300,fine,Ultrasonic_Cutter_TCP\WObj:=Workobject_2;
        MoveJ Con_850,v300,fine,Ultrasonic_Cutter_TCP\WObj:=Workobject_2;
        MoveJ Con_860,v300,fine,Ultrasonic_Cutter_TCP\WObj:=Workobject_2;
        MoveJ Target_30,v300,fine,Ultrasonic_Cutter_TCP\WObj:=Workobject_2;
        MoveJ Last_20,v300,z1,Ultrasonic_Cutter_TCP\WObj:=Workobject_2;
        MoveL Last_10,v300,z1,Ultrasonic_Cutter_TCP\WObj:=Workobject_2;
        MoveJ Target_80,v300,fine,Ultrasonic_Cutter_TCP\WObj:=Workobject_2;
        MoveJ Target_30,v300,fine,Ultrasonic_Cutter_TCP\WObj:=Workobject_2;
    ENDPROC
ENDMODULE
